# B&R Automation Studio project PLC code - cp
Automation Studio 4.1.4.357

## Configuration Dryer

CPU X20CP0483, AutomationRuntime G4.93, Build 4.1.2, Safety 0.0

### Task classes (Cpu.sw)
```
Cyclic#1 (cycle 8000 us, tolerance 8000 us):
  BasicDetec <- ExtPack._Media.BasicDetectMediaCtrl.BasicDetectMediaCtrl_v1.BasicDetectMediaCtrl.prg (BuildOptions=-D _IGNORE_CHECKLIB)
  ThickFast <- ExtPack._Media.ThicknessCtrl.ThicknessCtrl_v2.ThicknessCtrl_Fast.prg (BuildOptions=-D _IGNORE_CHECKLIB)
  VisuInks <- (binary) (BuildOptions=-D _IGNORE_CHECKLIB)
Cyclic#2 (cycle 12000 us, tolerance 24000 us):
  Initialize <- Dryer.Config.Initialize.prg (BuildOptions=-D _IGNORE_CHECKLIB)
  InitAxis <- ExtPack._Motion.AxisCtrl.AxisCtrl_v2.InitAxisControl.prg (BuildOptions=-D _IGNORE_CHECKLIB)
  Belt <- ExtPack._Motion.AxisCtrl.AxisCtrl_v2.AxisCtrl.prg (BuildOptions=-D _IGNORE_CHECKLIB)
  Elevation <- ExtPack._Motion.AxisCtrl.AxisCtrl_v2.AxisCtrl.prg (BuildOptions=-D _IGNORE_CHECKLIB)
  InitInvert <- ExtPack._Motion.InverterCtrl.InverterCtrl_v1.InitInverterCtrl.prg (BuildOptions=-D _IGNORE_CHECKLIB)
  Inverter1 <- ExtPack._Motion.InverterCtrl.InverterCtrl_v1.InverterCtrl.prg (BuildOptions=-D _IGNORE_CHECKLIB)
  Inverter2 <- ExtPack._Motion.InverterCtrl.InverterCtrl_v1.InverterCtrl.prg (BuildOptions=-D _IGNORE_CHECKLIB)
Cyclic#4 (cycle 32000 us, tolerance 96000 us):
  PhyInputs <- Dryer.PhysicalMapping.PhysicalMapInputs.prg (BuildOptions=-D _IGNORE_CHECKLIB)
  ThickCtrl <- ExtPack._Media.ThicknessCtrl.ThicknessCtrl_v2.ThicknessCtrl.prg (BuildOptions=-D _IGNORE_CHECKLIB)
  DryerFast <- Dryer.DryerCtrl.DryerCtrl_Fast.prg (BuildOptions=-D _IGNORE_CHECKLIB)
  BeltCtrl <- ExtPack._Transport.BeltCtrl.BeltCtrl_v1.BeltCtrl.prg (BuildOptions=-D _IGNORE_CHECKLIB)
  InitSimple <- ExtPack.SimpleBlockCtrl.SimpleBlockCtrl_v1.InitSimpleBlockCtrl.prg (BuildOptions=-D _IGNORE_CHECKLIB)
  SimpleBloc <- ExtPack.SimpleBlockCtrl.SimpleBlockCtrl_v1.SimpleBlockCtrl.prg (BuildOptions=-D _IGNORE_CHECKLIB)
  InitTransV <- ExtPack._Transport.TransVacuumCtrl.TransVacuumCtrl_v1.InitTransVacuumCtrl.prg (BuildOptions=-D _IGNORE_CHECKLIB)
  TransVacuu <- ExtPack._Transport.TransVacuumCtrl.TransVacuumCtrl_v1.TransVacuumCtrl.prg (BuildOptions=-D _IGNORE_CHECKLIB)
  InitJamDet <- ExtPack._Transport.JamDetectCtrl.JamDetect_v1.InitJamDetect.prg (BuildOptions=-D _IGNORE_CHECKLIB)
  JamDetect <- ExtPack._Transport.JamDetectCtrl.JamDetect_v1.JamDetect.prg (BuildOptions=-D _IGNORE_CHECKLIB)
  ArcLampGew <- ExtPack._Cure.ArcLampGEW.ArcLampGew_v1.ArcLampGewCtrl.prg (BuildOptions=-D _IGNORE_CHECKLIB)
  NIRAdphos <- ExtPack._Cure.NIRAdphos.NIRAdphos_v1.NIRAdphosCtrl.prg (BuildOptions=-D _IGNORE_CHECKLIB)
  HMI <- Dryer.HMI.HMI.prg (BuildOptions=-D _IGNORE_CHECKLIB)
  PhysOutput <- Dryer.PhysicalMapping.PhysicalMapOutputs.prg (BuildOptions=-D _IGNORE_CHECKLIB)
Cyclic#5 (cycle 80000 us, tolerance 160000 us):
  MachConfig <- Dryer.Config.MachineConfigurator.prg (BuildOptions=-D _IGNORE_CHECKLIB)
  DryerSlow <- Dryer.DryerCtrl.DryerCtrl_Slow.prg (BuildOptions=-D _IGNORE_CHECKLIB)
  ThickReadE <- ExtPack._Media.ThicknessCtrl.ThicknessCtrl_v2.ThickReadEnergy.prg (BuildOptions=-D _IGNORE_CHECKLIB)
  EventLogGe <- ExtPack._Tools.EventLog.EventLog_v1.EventLogGen.prg (BuildOptions=-D _IGNORE_CHECKLIB)
  SavePerman <- Dryer.Config.SavePermanent.prg (BuildOptions=-D _IGNORE_CHECKLIB)
NcDataObjects: AcpErrTxt <- AxisTables.AcpErrTxt.dob, acp10etxen <- AxisTables.acp10etxen.dob, BK1_S1400a <- AxisTables.BK1_S1400_a.dob, BK1_S1400i <- AxisTables.BK1_S1400_i.dob, BeltS1400a <- AxisTables.BeltS1400_a.dob, BeltS1400i <- AxisTables.BeltS1400_i.dob
Binaries: Acp10sys, udbdef, TCData, mvLoader, TCLang, arsvcreg, OpcUaSrv, acp10cfg, Acp10map, iomap, asfw, Role, ashwac, sysconf, ashwd, User, arconfig, EFIunits, EFIfunct, TC, gAlrHist, gAlrCore, OpcUaMap
Libraries: Acp10sdc, Acp10man, AsBrStr, Acp10par, NcGlobal, Acp10_MC, Acp10sim, sys_lib, brsystem, operator, runtime, astime, AsSafety, FileIO, standard, AsXml, asstring, AsFifo, MTTypes, MTFilter, MTBasics, AsTCP, AsIecCon, AsIOAcc, AsBrMath, AsEPL, ArEventLog, AsARCfg, ArProject, AsHttp, DataObj, FBs, Functions, ConvertFun, EvLogLib, BRSE_JSON, UtMgr, MpAlarmX, MpBase, MpCom, MpServer, AxisFunc, ThickLib, AsOpcUac, ErrACS380, arssl, aruser, powerlnk, assem, asopcuas, ascanopen
```

### Hardware
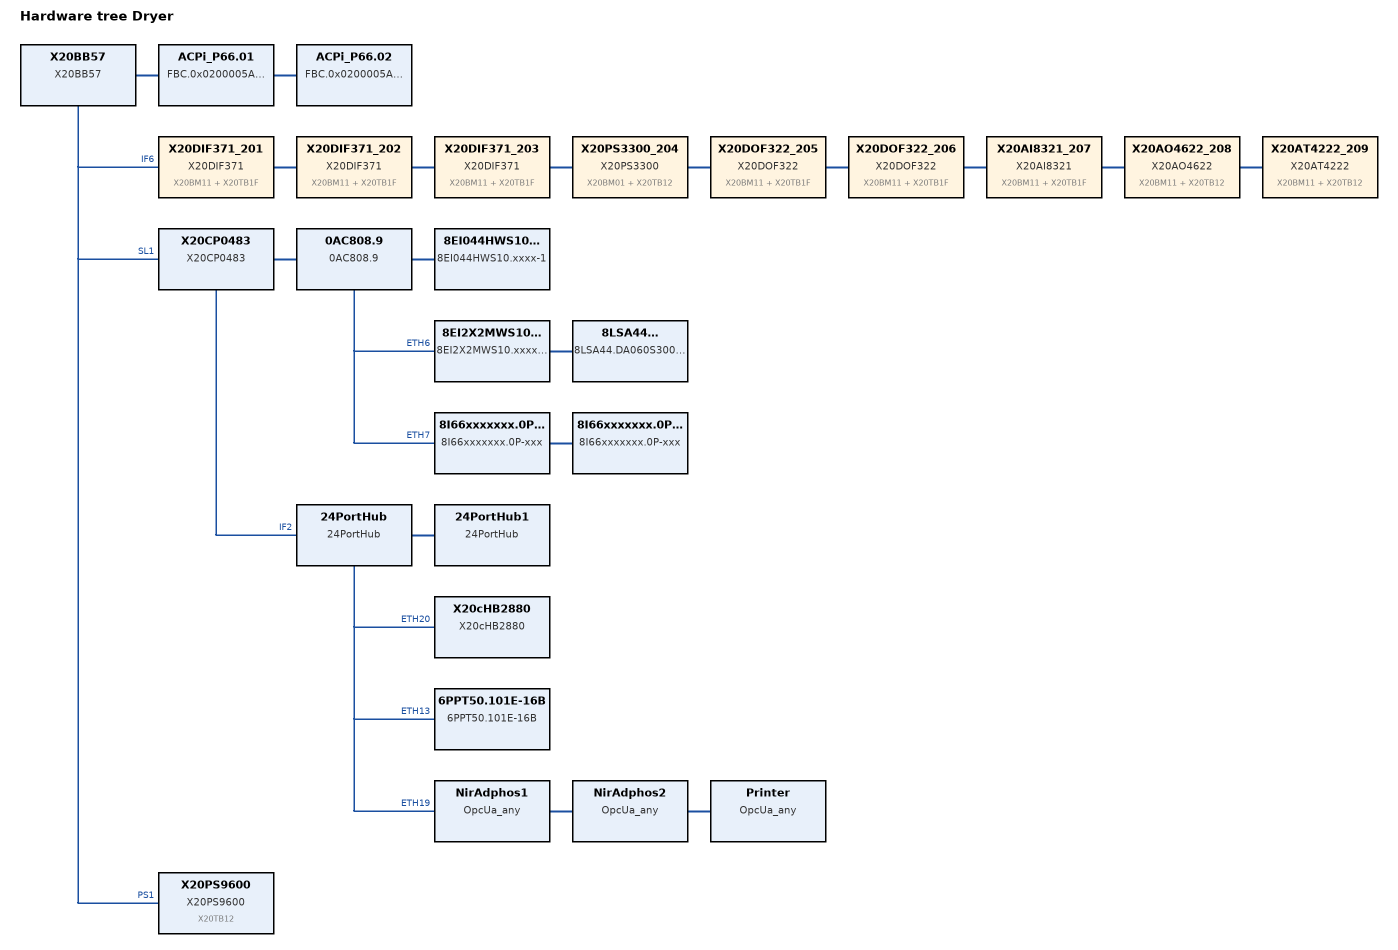
```
0AC808.9 : 0AC808.9 v1.0.0.0  [ETH1 -> X20CP0483.IF3 [Cable Type=PowerlinkCable, Length=10, Version=1.0.0.3]; ETH5 -> 8EI044HWS10.xxxx-1_BELT.PLK1 [Cable Type=PowerlinkCable, Length=10, Version=1.0.0.3]; ETH6 -> 8EI2X2MWS10.xxxx-1.PLK1 [Cable Type=PowerlinkCable, Length=10, Version=1.0.0.3]; ETH7 -> 8I66xxxxxxx.0P-81.PLK1 [Cable Type=PowerlinkCable, Length=10, Version=1.0.0.3]]
24PortHub : 24PortHub v1.0.0.1  [ETH7 -> X20CP0483.IF2 [Cable Type=PowerlinkCable, Length=10, Version=1.0.0.3]; ETH13 -> 6PPT50.101E-16B.ETH1 [Cable Type=PowerlinkCable, Length=10, Version=1.0.0.3]; ETH19 -> NirAdphos1.ETH1 [Cable Type=PowerlinkCable, Length=10, Version=1.0.0.3]; ETH20 -> X20cHB2880.ETH1 [Cable Type=PowerlinkCable, Length=10, Version=1.0.0.3]; ETH24 -> 24PortHub1.ETH3 [Cable Type=PowerlinkCable, Length=10, Version=1.0.0.3]]
24PortHub1 : 24PortHub v1.0.0.1  [ETH3 -> 24PortHub.ETH24 [Cable Type=PowerlinkCable, Length=10, Version=1.0.0.3]]
6PPT50.101E-16B : 6PPT50.101E-16B v1.3.8.0  [ETH1 -> 24PortHub.ETH13 [Cable Type=PowerlinkCable, Length=10, Version=1.0.0.3]]
  Terminal = true
  Startmode = 2
  ShowBootlogoWeb = 1
  Mode = Manual
  InternetAddress = 192.168.125.48
  Subnetmask = 255.255.255.0
  Hostname = efi_dryer_hmi
  Screensaver = 1
  Screensavertype = 0
  ActivateBuzzer = 1
  PasswordVNC = 
  SelectedFavoriteWeb = 192.168.125.47:81/index.html
  Favorites_Web1 = 
  BrowserVKeyboard = 0
  PasswordCIFS = 
  PasswordService = 
  ANSLAuthUserName = 
8EI044HWS10.xxxx-1_BELT : 8EI044HWS10.xxxx-1 v2.3.1.1  [PLK1 -> 0AC808.9.ETH5 [Cable Type=PowerlinkCable, Length=10, Version=1.0.0.3]]
  MotionTP = Acp10Arnc0
  Ax1Interface = Ax1EnDat
8EI2X2MWS10.xxxx-1 : 8EI2X2MWS10.xxxx-1 v2.3.1.1  [PLK1 -> 0AC808.9.ETH6 (NodeNumber=21) [Cable Type=PowerlinkCable, Length=10, Version=1.0.0.3]; EC1 -> 8LSA44.DA060S300-3.EC]
  MotionTP = Acp10Arnc0
  Ax1Interface = Ax1EnDat
8I66xxxxxxx.0P-81 : 8I66xxxxxxx.0P-xxx v2.5.1.0  [PLK1 -> 0AC808.9.ETH7 (NodeNumber=81) [Cable Type=PowerlinkCable, Length=10, Version=1.0.0.3]; PLK2 -> 8I66xxxxxxx.0P-82.PLK1 (NodeNumber=81) [Cable Type=PowerlinkCable, Length=10, Version=1.0.0.3]]
  FunctionModel = Standard
  Supervision = off
  UnitOfSetpoint = Rpm
  IOM_AIDP1 = LFT
  IOM_AIDP2 = LCR
  IOM_AIDP3 = OTRN
  IOM_AIDP4 = IL1R
  IOM_AIDP5 = AI1R
  IOM_AIDP6 = AI2R
  IOM_AIDP7 = AI3R
  IOM_AIDP8 = OL1I
  IOM_AIDP9 = AO1I
  IOM_R1ctrl = mapped
  IOM_R2ctrl = mapped
  IOM_LO1ctrl = mapped
  IOM_AO1ctrl = mapped
  Sel_AO1T = 0A
  Sel_NameplateMask = 8Ix6T401500_IEC
  Cfg_NSP = 2940
  Cfg_NCR = 277
  Cfg_COS = 82
  Sel_TUN = AUTO
8I66xxxxxxx.0P-82 : 8I66xxxxxxx.0P-xxx v2.5.1.0  [PLK1 -> 8I66xxxxxxx.0P-81.PLK2 [Cable Type=PowerlinkCable, Length=10, Version=1.0.0.3]]
  FunctionModel = Standard
  Supervision = off
  UnitOfSetpoint = Rpm
  IOM_AIDP1 = LFT
  IOM_AIDP2 = LCR
  IOM_AIDP3 = OTRN
  IOM_AIDP4 = IL1R
  IOM_AIDP5 = AI1R
  IOM_AIDP6 = AI2R
  IOM_AIDP7 = AI3R
  IOM_AIDP8 = OL1I
  IOM_AIDP9 = AO1I
  IOM_R1ctrl = mapped
  IOM_R2ctrl = mapped
  IOM_LO1ctrl = mapped
  IOM_AO1ctrl = mapped
  Sel_AO1T = 0A
  Sel_NameplateMask = 8Ix6T401500_IEC
  Cfg_NSP = 2940
  Cfg_NCR = 277
  Cfg_COS = 82
  Sel_TUN = AUTO
8LSA44.DA060S300-3 : 8LSA44.DA060S300-3 v1.0.10.37  [EC -> 8EI2X2MWS10.xxxx-1.EC1; MT -> 8EI2X2MWS10.xxxx-1.MT1]
ACPi_P66.01 : FBC.0x0200005A.320.ACPi_P66_P76 v1.3 (OrderNumber=ACPi_P66_P76)  [CAN1 -> X20BB57.IF7 (NodeNumber=81)]
  p2002sub5_connecttomaster = 2
  p2016sub3_connecttomaster = 1
  p2016subd_connecttomaster = 5
  p2016sub21_connecttomaster = 1
  p2016sub22_connecttomaster = 1
  p2016sub3e_connecttomaster = 5
  p2029sub16_connecttomaster = 2
  p2038sub2_connecttomaster = 4
  p2038sub3_connecttomaster = 4
  p2038sub4_connecttomaster = 2
  p2038sub5_connecttomaster = 2
  p203csub2_connecttomaster = 5
  p203csub3_connecttomaster = 5
  p6040_connecttomaster = 0
  p6041_connecttomaster = 0
  p6042_connecttomaster = 0
  p6044_connecttomaster = 0
  p6077_connecttomaster = 1
  p1800_transmissionselection = 2
  p1801_transmissionselection = 2
  p1802_transmissionselection = 2
ACPi_P66.02 : FBC.0x0200005A.320.ACPi_P66_P76 v1.3 (OrderNumber=ACPi_P66_P76)  [CAN1 -> ACPi_P66.01.CAN2]
  p2002sub5_connecttomaster = 2
  p2016sub3_connecttomaster = 1
  p2016subd_connecttomaster = 5
  p2016sub21_connecttomaster = 1
  p2016sub22_connecttomaster = 1
  p2016sub3e_connecttomaster = 5
  p2029sub16_connecttomaster = 2
  p2038sub2_connecttomaster = 4
  p2038sub3_connecttomaster = 4
  p2038sub4_connecttomaster = 2
  p2038sub5_connecttomaster = 2
  p203csub2_connecttomaster = 5
  p203csub3_connecttomaster = 5
  p6040_connecttomaster = 0
  p6041_connecttomaster = 0
  p6042_connecttomaster = 0
  p6044_connecttomaster = 0
  p6077_connecttomaster = 1
  p1800_transmissionselection = 2
  p1801_transmissionselection = 2
  p1802_transmissionselection = 2
NirAdphos1 : OpcUa_any v1.0.0.1  [ETH1 -> 24PortHub.ETH19 [Cable Type=PowerlinkCable, Length=10, Version=1.0.0.3]; ETH2 -> NirAdphos2.ETH1 [Cable Type=PowerlinkCable, Length=10, Version=1.0.0.3]]
  ServerDiagnostics = on
  ServerEndpointUrl = opc.tcp://192.168.125.91:4840
  PnPTimeout = 2500
  SecurityMsgMode = 0
  Channel1
  ChannelID1 = HMI
  ChannelBrowsePath1 = /0:Root/0:Objects/3:ServerInterfaces/4:SendData/4:DB11_HMI_out/4:HMI
  ChannelType1 = INT
  Channel2
  ChannelID2 = Hardware
  ChannelBrowsePath2 = /0:Root/0:Objects/3:ServerInterfaces/4:SendData/4:DB11_HMI_out/4:Hardware
  ChannelType2 = INT
  Channel3
  ChannelID3 = Software
  ChannelBrowsePath3 = /0:Root/0:Objects/3:ServerInterfaces/4:SendData/4:DB11_HMI_out/4:Software
  ChannelType3 = INT
  Channel4
  ChannelID4 = Interface
  ChannelBrowsePath4 = /0:Root/0:Objects/3:ServerInterfaces/4:SendData/4:DB11_HMI_out/4:interface
  ChannelType4 = INT
  Channel5
  ChannelID5 = NIRno
  ChannelBrowsePath5 = /0:Root/0:Objects/3:ServerInterfaces/4:SendData/4:DB11_HMI_out/4:general/4:NIRno
  ChannelType5 = INT
  Channel6
  ChannelID6 = NIRwidth
  ChannelBrowsePath6 = /0:Root/0:Objects/3:ServerInterfaces/4:SendData/4:DB11_HMI_out/4:general/4:NIRwidth
  ChannelType6 = INT
  Channel7
  ChannelID7 = calPower
  ChannelBrowsePath7 = /0:Root/0:Objects/3:ServerInterfaces/4:SendData/4:DB11_HMI_out/4:general/4:calPower
  ChannelType7 = INT
  Channel8
  ChannelID8 = speed
  ChannelBrowsePath8 = /0:Root/0:Objects/3:ServerInterfaces/4:SendData/4:DB11_HMI_out/4:general/4:speed
  ChannelType8 = REAL
  Channel9
  ChannelID9 = Watchdog1
  ChannelBrowsePath9 = /0:Root/0:Objects/3:ServerInterfaces/4:SendData/4:DB11_HMI_out/4:general/4:Watchdog
  Channel10
  ChannelID10 = EmFailNo_1
  ChannelBrowsePath10 = /0:Root/0:Objects/3:ServerInterfaces/4:SendData/4:DB11_HMI_out/4:module/4:[1]/4:EmFailNo
  ChannelType10 = USINT
  Channel11
  ChannelID11 = EmFailNo_2
  ChannelBrowsePath11 = /0:Root/0:Objects/3:ServerInterfaces/4:SendData/4:DB11_HMI_out/4:module/4:[2]/4:EmFailNo
  ChannelType11 = USINT
  Channel12
  ChannelID12 = ExhAirRunning_1
  ChannelBrowsePath12 = /0:Root/0:Objects/3:ServerInterfaces/4:SendData/4:DB11_HMI_out/4:module/4:[1]/4:ExhAirRunning
  Channel13
  ChannelID13 = ExhAirRunning_2
  ChannelBrowsePath13 = /0:Root/0:Objects/3:ServerInterfaces/4:SendData/4:DB11_HMI_out/4:module/4:[2]/4:ExhAirRunning
  Channel14
  ChannelID14 = NIRstatus_1
  ChannelBrowsePath14 = /0:Root/0:Objects/3:ServerInterfaces/4:SendData/4:DB11_HMI_out/4:module/4:[1]/4:NIRstatus
  ChannelType14 = INT
  Channel15
  ChannelID15 = NIRstatus_2
  ChannelBrowsePath15 = /0:Root/0:Objects/3:ServerInterfaces/4:SendData/4:DB11_HMI_out/4:module/4:[2]/4:NIRstatus
  ChannelType15 = INT
  Channel16
  ChannelID16 = airPressIn_1
  ChannelBrowsePath16 = /0:Root/0:Objects/3:ServerInterfaces/4:SendData/4:DB11_HMI_out/4:module/4:[1]/4:airPressIn
  ChannelType16 = REAL
  Channel17
  ChannelID17 = airPressIn_2
  ChannelBrowsePath17 = /0:Root/0:Objects/3:ServerInterfaces/4:SendData/4:DB11_HMI_out/4:module/4:[2]/4:airPressIn
  ChannelType17 = REAL
  Channel18
  ChannelID18 = airPressOut_1
  ChannelBrowsePath18 = /0:Root/0:Objects/3:ServerInterfaces/4:SendData/4:DB11_HMI_out/4:module/4:[1]/4:airPressOut
  ChannelType18 = REAL
  Channel19
  ChannelID19 = airPressOut_2
  ChannelBrowsePath19 = /0:Root/0:Objects/3:ServerInterfaces/4:SendData/4:DB11_HMI_out/4:module/4:[2]/4:airPressOut
  ChannelType19 = REAL
  Channel20
  ChannelID20 = airFilter_1
  ChannelBrowsePath20 = /0:Root/0:Objects/3:ServerInterfaces/4:SendData/4:DB11_HMI_out/4:module/4:[1]/4:airFilter
  ChannelType20 = INT
  Channel21
  ChannelID21 = airFilter_2
  ChannelBrowsePath21 = /0:Root/0:Objects/3:ServerInterfaces/4:SendData/4:DB11_HMI_out/4:module/4:[2]/4:airFilter
  ChannelType21 = INT
  Channel22
  ChannelID22 = actSpeedIn_1
  ChannelBrowsePath22 = /0:Root/0:Objects/3:ServerInterfaces/4:SendData/4:DB11_HMI_out/4:module/4:[1]/4:actSpeedIn
  ChannelType22 = INT
  Channel23
  ChannelID23 = actSpeedIn_2
  ChannelBrowsePath23 = /0:Root/0:Objects/3:ServerInterfaces/4:SendData/4:DB11_HMI_out/4:module/4:[2]/4:actSpeedIn
  ChannelType23 = INT
  Channel24
  ChannelID24 = actSpeedOut_1
  ChannelBrowsePath24 = /0:Root/0:Objects/3:ServerInterfaces/4:SendData/4:DB11_HMI_out/4:module/4:[1]/4:actSpeedOut
  ChannelType24 = INT
  Channel25
  ChannelID25 = actSpeedOut_2
  ChannelBrowsePath25 = /0:Root/0:Objects/3:ServerInterfaces/4:SendData/4:DB11_HMI_out/4:module/4:[2]/4:actSpeedOut
  ChannelType25 = INT
  Channel26
  ChannelID26 = actPower_1
  ChannelBrowsePath26 = /0:Root/0:Objects/3:ServerInterfaces/4:SendData/4:DB11_HMI_out/4:module/4:[1]/4:actPower
  ChannelType26 = INT
  Channel27
  ChannelID27 = actPower_2
  ChannelBrowsePath27 = /0:Root/0:Objects/3:ServerInterfaces/4:SendData/4:DB11_HMI_out/4:module/4:[2]/4:actPower
  ChannelType27 = INT
  Channel28
  ChannelID28 = Watchdog2
  ChannelBrowsePath28 = /0:Root/0:Objects/3:ServerInterfaces/4:SendData/4:DB11_HMI_out/4:general/4:Watchdog
  Channel29
  ChannelID29 = Reset
  ChannelBrowsePath29 = /0:Root/0:Objects/3:ServerInterfaces/5:RecData/5:DB10_HMI_in/5:reset
  ChannelDirection29 = OUT
  Channel30
  ChannelID30 = Pend
  ChannelBrowsePath30 = /0:Root/0:Objects/3:ServerInterfaces/5:RecData/5:DB10_HMI_in/5:product/5:Pend
  ChannelDirection30 = OUT
  ChannelType30 = REAL
  Channel31
  ChannelID31 = Pstart
  ChannelBrowsePath31 = /0:Root/0:Objects/3:ServerInterfaces/5:RecData/5:DB10_HMI_in/5:product/5:Pstart
  ChannelDirection31 = OUT
  ChannelType31 = REAL
  Channel32
  ChannelID32 = Vend
  ChannelBrowsePath32 = /0:Root/0:Objects/3:ServerInterfaces/5:RecData/5:DB10_HMI_in/5:product/5:Vend
  ChannelDirection32 = OUT
  ChannelType32 = REAL
  Channel33
  ChannelID33 = Vstart
  ChannelBrowsePath33 = /0:Root/0:Objects/3:ServerInterfaces/5:RecData/5:DB10_HMI_in/5:product/5:Vstart
  ChannelDirection33 = OUT
  ChannelType33 = REAL
  Channel34
  ChannelID34 = AdjPos
  ChannelBrowsePath34 = /0:Root/0:Objects/3:ServerInterfaces/5:RecData/5:DB10_HMI_in/5:product/5:adjPos
  ChannelDirection34 = OUT
  ChannelType34 = INT
  Channel35
  ChannelID35 = WebWidth
  ChannelBrowsePath35 = /0:Root/0:Objects/3:ServerInterfaces/5:RecData/5:DB10_HMI_in/5:product/5:webWidth
  ChannelDirection35 = OUT
  ChannelType35 = INT
  Channel36
  ChannelID36 = Adjust_1
  ChannelBrowsePath36 = /0:Root/0:Objects/3:ServerInterfaces/5:RecData/5:DB10_HMI_in/5:module/5:[1]/5:adjust
  ChannelDirection36 = OUT
  ChannelType36 = INT
  Channel37
  ChannelID37 = Adjust_2
  ChannelBrowsePath37 = /0:Root/0:Objects/3:ServerInterfaces/5:RecData/5:DB10_HMI_in/5:module/5:[2]/5:adjust
  ChannelDirection37 = OUT
  ChannelType37 = INT
  Channel38
  ChannelID38 = EnableMod_1
  ChannelBrowsePath38 = /0:Root/0:Objects/3:ServerInterfaces/5:RecData/5:DB10_HMI_in/5:module/5:[1]/5:enableMod
  ChannelDirection38 = OUT
  Channel39
  ChannelID39 = EnableMod_2
  ChannelBrowsePath39 = /0:Root/0:Objects/3:ServerInterfaces/5:RecData/5:DB10_HMI_in/5:module/5:[2]/5:enableMod
  ChannelDirection39 = OUT
  Channel40
  ChannelID40 = WatchdogOut
  ChannelBrowsePath40 = /0:Root/0:Objects/3:ServerInterfaces/5:RecData/5:DB10_HMI_in/5:Watchdog
  ChannelDirection40 = OUT
  Channel41
  ChannelID41 = Enable_DDC
  ChannelBrowsePath41 = /0:Root/0:Objects/3:ServerInterfaces/5:RecData/5:DB10_HMI_in/5:DDCon
  ChannelDirection41 = OUT
  Channel42
  ChannelID42 = NIR1_Int1
  ChannelBrowsePath42 = /0:Root/0:Objects/3:ServerInterfaces/5:RecData/5:DB10_HMI_in/5:intensity/5:intensity/5:[1]
  ChannelDirection42 = OUT
  ChannelType42 = INT
  Channel43
  ChannelID43 = NIR1_Int2
  ChannelBrowsePath43 = /0:Root/0:Objects/3:ServerInterfaces/5:RecData/5:DB10_HMI_in/5:intensity/5:intensity/5:[2]
  ChannelDirection43 = OUT
  ChannelType43 = INT
  Channel44
  ChannelID44 = NIR1_Int3
  ChannelBrowsePath44 = /0:Root/0:Objects/3:ServerInterfaces/5:RecData/5:DB10_HMI_in/5:intensity/5:intensity/5:[3]
  ChannelDirection44 = OUT
  ChannelType44 = INT
  Channel45
  ChannelID45 = NIR1_Int4
  ChannelBrowsePath45 = /0:Root/0:Objects/3:ServerInterfaces/5:RecData/5:DB10_HMI_in/5:intensity/5:intensity/5:[4]
  ChannelDirection45 = OUT
  ChannelType45 = INT
  Channel46
  ChannelID46 = NIR1_Int5
  ChannelBrowsePath46 = /0:Root/0:Objects/3:ServerInterfaces/5:RecData/5:DB10_HMI_in/5:intensity/5:intensity/5:[5]
  ChannelDirection46 = OUT
  ChannelType46 = INT
  Channel47
  ChannelID47 = NIR1_Int6
  ChannelBrowsePath47 = /0:Root/0:Objects/3:ServerInterfaces/5:RecData/5:DB10_HMI_in/5:intensity/5:intensity/5:[6]
  ChannelDirection47 = OUT
  ChannelType47 = INT
  Channel48
  ChannelID48 = NIR1_Int7
  ChannelBrowsePath48 = /0:Root/0:Objects/3:ServerInterfaces/5:RecData/5:DB10_HMI_in/5:intensity/5:intensity/5:[7]
  ChannelDirection48 = OUT
  ChannelType48 = INT
  Channel49
  ChannelID49 = NIR1_Int8
  ChannelBrowsePath49 = /0:Root/0:Objects/3:ServerInterfaces/5:RecData/5:DB10_HMI_in/5:intensity/5:intensity/5:[8]
  ChannelDirection49 = OUT
  ChannelType49 = INT
  Channel50
  ChannelID50 = NIR1_Int9
  ChannelBrowsePath50 = /0:Root/0:Objects/3:ServerInterfaces/5:RecData/5:DB10_HMI_in/5:intensity/5:intensity/5:[9]
  ChannelDirection50 = OUT
  ChannelType50 = INT
  Channel51
  ChannelID51 = NIR1_Int10
  ChannelBrowsePath51 = /0:Root/0:Objects/3:ServerInterfaces/5:RecData/5:DB10_HMI_in/5:intensity/5:intensity/5:[10]
  ChannelDirection51 = OUT
  ChannelType51 = INT
  Channel52
  ChannelID52 = NIR1_Int11
  ChannelBrowsePath52 = /0:Root/0:Objects/3:ServerInterfaces/5:RecData/5:DB10_HMI_in/5:intensity/5:intensity/5:[11]
  ChannelDirection52 = OUT
  ChannelType52 = INT
  Channel53
  ChannelID53 = NIR1_Int12
  ChannelBrowsePath53 = /0:Root/0:Objects/3:ServerInterfaces/5:RecData/5:DB10_HMI_in/5:intensity/5:intensity/5:[12]
  ChannelDirection53 = OUT
  ChannelType53 = INT
  Channel54
  ChannelID54 = NIR1_Int13
  ChannelBrowsePath54 = /0:Root/0:Objects/3:ServerInterfaces/5:RecData/5:DB10_HMI_in/5:intensity/5:intensity/5:[13]
  ChannelDirection54 = OUT
  ChannelType54 = INT
  Channel55
  ChannelID55 = NIR1_Int14
  ChannelBrowsePath55 = /0:Root/0:Objects/3:ServerInterfaces/5:RecData/5:DB10_HMI_in/5:intensity/5:intensity/5:[14]
  ChannelDirection55 = OUT
  ChannelType55 = INT
  Channel56
  ChannelID56 = NIR1_Int15
  ChannelBrowsePath56 = /0:Root/0:Objects/3:ServerInterfaces/5:RecData/5:DB10_HMI_in/5:intensity/5:intensity/5:[15]
  ChannelDirection56 = OUT
  ChannelType56 = INT
  Channel57
  ChannelID57 = NIR1_Int16
  ChannelBrowsePath57 = /0:Root/0:Objects/3:ServerInterfaces/5:RecData/5:DB10_HMI_in/5:intensity/5:intensity/5:[16]
  ChannelDirection57 = OUT
  ChannelType57 = INT
  Channel58
  ChannelID58 = NIR1_Int17
  ChannelBrowsePath58 = /0:Root/0:Objects/3:ServerInterfaces/5:RecData/5:DB10_HMI_in/5:intensity/5:intensity/5:[17]
  ChannelDirection58 = OUT
  ChannelType58 = INT
  Channel59
  ChannelID59 = NIR1_Int18
  ChannelBrowsePath59 = /0:Root/0:Objects/3:ServerInterfaces/5:RecData/5:DB10_HMI_in/5:intensity/5:intensity/5:[18]
  ChannelDirection59 = OUT
  ChannelType59 = INT
  Channel60
  ChannelID60 = NIR1_Int19
  ChannelBrowsePath60 = /0:Root/0:Objects/3:ServerInterfaces/5:RecData/5:DB10_HMI_in/5:intensity/5:intensity/5:[19]
  ChannelDirection60 = OUT
  ChannelType60 = INT
  Channel61
  ChannelID61 = NIR1_Int20
  ChannelBrowsePath61 = /0:Root/0:Objects/3:ServerInterfaces/5:RecData/5:DB10_HMI_in/5:intensity/5:intensity/5:[20]
  ChannelDirection61 = OUT
  ChannelType61 = INT
  Channel62
  ChannelID62 = NIR1_Int21
  ChannelBrowsePath62 = /0:Root/0:Objects/3:ServerInterfaces/5:RecData/5:DB10_HMI_in/5:intensity/5:intensity/5:[21]
  ChannelDirection62 = OUT
  ChannelType62 = INT
  Channel63
  ChannelID63 = NIR1_Int22
  ChannelBrowsePath63 = /0:Root/0:Objects/3:ServerInterfaces/5:RecData/5:DB10_HMI_in/5:intensity/5:intensity/5:[22]
  ChannelDirection63 = OUT
  ChannelType63 = INT
  Channel64
  ChannelID64 = NIR1_Int23
  ChannelBrowsePath64 = /0:Root/0:Objects/3:ServerInterfaces/5:RecData/5:DB10_HMI_in/5:intensity/5:intensity/5:[23]
  ChannelDirection64 = OUT
  ChannelType64 = INT
  Channel65
  ChannelID65 = NIR1_Int24
  ChannelBrowsePath65 = /0:Root/0:Objects/3:ServerInterfaces/5:RecData/5:DB10_HMI_in/5:intensity/5:intensity/5:[24]
  ChannelDirection65 = OUT
  ChannelType65 = INT
  Channel66
  ChannelID66 = NIR1_Int25
  ChannelBrowsePath66 = /0:Root/0:Objects/3:ServerInterfaces/5:RecData/5:DB10_HMI_in/5:intensity/5:intensity/5:[25]
  ChannelDirection66 = OUT
  ChannelType66 = INT
  Channel67
  ChannelID67 = NIR1_Int26
  ChannelBrowsePath67 = /0:Root/0:Objects/3:ServerInterfaces/5:RecData/5:DB10_HMI_in/5:intensity/5:intensity/5:[26]
  ChannelDirection67 = OUT
  ChannelType67 = INT
  Channel68
  ChannelID68 = NIR1_Int27
  ChannelBrowsePath68 = /0:Root/0:Objects/3:ServerInterfaces/5:RecData/5:DB10_HMI_in/5:intensity/5:intensity/5:[27]
  ChannelDirection68 = OUT
  ChannelType68 = INT
  Channel69
  ChannelID69 = NIR1_Int28
  ChannelBrowsePath69 = /0:Root/0:Objects/3:ServerInterfaces/5:RecData/5:DB10_HMI_in/5:intensity/5:intensity/5:[28]
  ChannelDirection69 = OUT
  ChannelType69 = INT
  Channel70
  ChannelID70 = NIR1_Int29
  ChannelBrowsePath70 = /0:Root/0:Objects/3:ServerInterfaces/5:RecData/5:DB10_HMI_in/5:intensity/5:intensity/5:[29]
  ChannelDirection70 = OUT
  ChannelType70 = INT
  Channel71
  ChannelID71 = NIR1_Int30
  ChannelBrowsePath71 = /0:Root/0:Objects/3:ServerInterfaces/5:RecData/5:DB10_HMI_in/5:intensity/5:intensity/5:[30]
  ChannelDirection71 = OUT
  ChannelType71 = INT
  Channel72
  ChannelID72 = NIR1_Int31
  ChannelBrowsePath72 = /0:Root/0:Objects/3:ServerInterfaces/5:RecData/5:DB10_HMI_in/5:intensity/5:intensity/5:[31]
  ChannelDirection72 = OUT
  ChannelType72 = INT
  Channel73
  ChannelID73 = NIR1_Int32
  ChannelBrowsePath73 = /0:Root/0:Objects/3:ServerInterfaces/5:RecData/5:DB10_HMI_in/5:intensity/5:intensity/5:[32]
  ChannelDirection73 = OUT
  ChannelType73 = INT
  Channel74
  ChannelID74 = NIR1_Int33
  ChannelBrowsePath74 = /0:Root/0:Objects/3:ServerInterfaces/5:RecData/5:DB10_HMI_in/5:intensity/5:intensity/5:[33]
  ChannelDirection74 = OUT
  ChannelType74 = INT
  Channel75
  ChannelID75 = NIR1_Int34
  ChannelBrowsePath75 = /0:Root/0:Objects/3:ServerInterfaces/5:RecData/5:DB10_HMI_in/5:intensity/5:intensity/5:[34]
  ChannelDirection75 = OUT
  ChannelType75 = INT
  Channel76
  ChannelID76 = NIR1_Int35
  ChannelBrowsePath76 = /0:Root/0:Objects/3:ServerInterfaces/5:RecData/5:DB10_HMI_in/5:intensity/5:intensity/5:[35]
  ChannelDirection76 = OUT
  ChannelType76 = INT
  Channel77
  ChannelID77 = NIR1_Int36
  ChannelBrowsePath77 = /0:Root/0:Objects/3:ServerInterfaces/5:RecData/5:DB10_HMI_in/5:intensity/5:intensity/5:[36]
  ChannelDirection77 = OUT
  ChannelType77 = INT
  Channel78
  ChannelID78 = NIR1_Int37
  ChannelBrowsePath78 = /0:Root/0:Objects/3:ServerInterfaces/5:RecData/5:DB10_HMI_in/5:intensity/5:intensity/5:[37]
  ChannelDirection78 = OUT
  ChannelType78 = INT
  Channel79
  ChannelID79 = NIR1_Int38
  ChannelBrowsePath79 = /0:Root/0:Objects/3:ServerInterfaces/5:RecData/5:DB10_HMI_in/5:intensity/5:intensity/5:[38]
  ChannelDirection79 = OUT
  ChannelType79 = INT
  Channel80
  ChannelID80 = NIR1_Int39
  ChannelBrowsePath80 = /0:Root/0:Objects/3:ServerInterfaces/5:RecData/5:DB10_HMI_in/5:intensity/5:intensity/5:[39]
  ChannelDirection80 = OUT
  ChannelType80 = INT
  Channel81
  ChannelID81 = NIR1_Int40
  ChannelBrowsePath81 = /0:Root/0:Objects/3:ServerInterfaces/5:RecData/5:DB10_HMI_in/5:intensity/5:intensity/5:[40]
  ChannelDirection81 = OUT
  ChannelType81 = INT
  Channel82
  ChannelID82 = NIR1_Int41
  ChannelBrowsePath82 = /0:Root/0:Objects/3:ServerInterfaces/5:RecData/5:DB10_HMI_in/5:intensity/5:intensity/5:[41]
  ChannelDirection82 = OUT
  ChannelType82 = INT
  Channel83
  ChannelID83 = NIR1_Int42
  ChannelBrowsePath83 = /0:Root/0:Objects/3:ServerInterfaces/5:RecData/5:DB10_HMI_in/5:intensity/5:intensity/5:[42]
  ChannelDirection83 = OUT
  ChannelType83 = INT
  Channel84
  ChannelID84 = NIR1_Int43
  ChannelBrowsePath84 = /0:Root/0:Objects/3:ServerInterfaces/5:RecData/5:DB10_HMI_in/5:intensity/5:intensity/5:[43]
  ChannelDirection84 = OUT
  ChannelType84 = INT
  Channel85
  ChannelID85 = NIR1_Int44
  ChannelBrowsePath85 = /0:Root/0:Objects/3:ServerInterfaces/5:RecData/5:DB10_HMI_in/5:intensity/5:intensity/5:[44]
  ChannelDirection85 = OUT
  ChannelType85 = INT
  Channel86
  ChannelID86 = NIR1_Int45
  ChannelBrowsePath86 = /0:Root/0:Objects/3:ServerInterfaces/5:RecData/5:DB10_HMI_in/5:intensity/5:intensity/5:[45]
  ChannelDirection86 = OUT
  ChannelType86 = INT
  Channel87
  ChannelID87 = NIR1_Int46
  ChannelBrowsePath87 = /0:Root/0:Objects/3:ServerInterfaces/5:RecData/5:DB10_HMI_in/5:intensity/5:intensity/5:[46]
  ChannelDirection87 = OUT
  ChannelType87 = INT
  Channel88
  ChannelID88 = NIR1_Int47
  ChannelBrowsePath88 = /0:Root/0:Objects/3:ServerInterfaces/5:RecData/5:DB10_HMI_in/5:intensity/5:intensity/5:[47]
  ChannelDirection88 = OUT
  ChannelType88 = INT
  Channel89
  ChannelID89 = NIR1_Int48
  ChannelBrowsePath89 = /0:Root/0:Objects/3:ServerInterfaces/5:RecData/5:DB10_HMI_in/5:intensity/5:intensity/5:[48]
  ChannelDirection89 = OUT
  ChannelType89 = INT
NirAdphos2 : OpcUa_any v1.0.0.1  [ETH1 -> NirAdphos1.ETH2 [Cable Type=PowerlinkCable, Length=10, Version=1.0.0.3]; ETH2 -> Printer.ETH1 [Cable Type=PowerlinkCable, Length=10, Version=1.0.0.3]]
  ServerDiagnostics = on
  ServerEndpointUrl = opc.tcp://192.168.125.92:4840
  PnPTimeout = 2500
  SecurityMsgMode = 0
  Channel1
  ChannelID1 = NIR2_Int1
  ChannelBrowsePath1 = /0:Root/0:Objects/3:ServerInterfaces/0:RecData/4:DB10_HMI_in/4:intensity/4:[1]
  ChannelDirection1 = OUT
  ChannelType1 = INT
  Channel2
  ChannelID2 = NIR2_Int2
  ChannelBrowsePath2 = /0:Root/0:Objects/3:ServerInterfaces/0:RecData/4:DB10_HMI_in/4:intensity/4:[2]
  ChannelDirection2 = OUT
  ChannelType2 = INT
  Channel3
  ChannelID3 = NIR2_Int3
  ChannelBrowsePath3 = /0:Root/0:Objects/3:ServerInterfaces/0:RecData/4:DB10_HMI_in/4:intensity/4:[3]
  ChannelDirection3 = OUT
  ChannelType3 = INT
  Channel4
  ChannelID4 = NIR2_Int4
  ChannelBrowsePath4 = /0:Root/0:Objects/3:ServerInterfaces/0:RecData/4:DB10_HMI_in/4:intensity/4:[4]
  ChannelDirection4 = OUT
  ChannelType4 = INT
  Channel5
  ChannelID5 = NIR2_Int5
  ChannelBrowsePath5 = /0:Root/0:Objects/3:ServerInterfaces/0:RecData/4:DB10_HMI_in/4:intensity/4:[5]
  ChannelDirection5 = OUT
  ChannelType5 = INT
  Channel6
  ChannelID6 = NIR2_Int6
  ChannelBrowsePath6 = /0:Root/0:Objects/3:ServerInterfaces/0:RecData/4:DB10_HMI_in/4:intensity/4:[6]
  ChannelDirection6 = OUT
  ChannelType6 = INT
  Channel7
  ChannelID7 = NIR2_Int7
  ChannelBrowsePath7 = /0:Root/0:Objects/3:ServerInterfaces/0:RecData/4:DB10_HMI_in/4:intensity/4:[7]
  ChannelDirection7 = OUT
  ChannelType7 = INT
  Channel8
  ChannelID8 = NIR2_Int8
  ChannelBrowsePath8 = /0:Root/0:Objects/3:ServerInterfaces/0:RecData/4:DB10_HMI_in/4:intensity/4:[8]
  ChannelDirection8 = OUT
  ChannelType8 = INT
  Channel9
  ChannelID9 = NIR2_Int9
  ChannelBrowsePath9 = /0:Root/0:Objects/3:ServerInterfaces/0:RecData/4:DB10_HMI_in/4:intensity/4:[9]
  ChannelDirection9 = OUT
  ChannelType9 = INT
  Channel10
  ChannelID10 = NIR2_Int10
  ChannelBrowsePath10 = /0:Root/0:Objects/3:ServerInterfaces/0:RecData/4:DB10_HMI_in/4:intensity/4:[10]
  ChannelDirection10 = OUT
  ChannelType10 = INT
  Channel11
  ChannelID11 = NIR2_Int11
  ChannelBrowsePath11 = /0:Root/0:Objects/3:ServerInterfaces/0:RecData/4:DB10_HMI_in/4:intensity/4:[11]
  ChannelDirection11 = OUT
  ChannelType11 = INT
  Channel12
  ChannelID12 = NIR2_Int12
  ChannelBrowsePath12 = /0:Root/0:Objects/3:ServerInterfaces/0:RecData/4:DB10_HMI_in/4:intensity/4:[12]
  ChannelDirection12 = OUT
  ChannelType12 = INT
  Channel13
  ChannelID13 = NIR2_Int13
  ChannelBrowsePath13 = /0:Root/0:Objects/3:ServerInterfaces/0:RecData/4:DB10_HMI_in/4:intensity/4:[13]
  ChannelDirection13 = OUT
  ChannelType13 = INT
  Channel14
  ChannelID14 = NIR2_Int14
  ChannelBrowsePath14 = /0:Root/0:Objects/3:ServerInterfaces/0:RecData/4:DB10_HMI_in/4:intensity/4:[14]
  ChannelDirection14 = OUT
  ChannelType14 = INT
  Channel15
  ChannelID15 = NIR2_Int15
  ChannelBrowsePath15 = /0:Root/0:Objects/3:ServerInterfaces/0:RecData/4:DB10_HMI_in/4:intensity/4:[15]
  ChannelDirection15 = OUT
  ChannelType15 = INT
  Channel16
  ChannelID16 = NIR2_Int16
  ChannelBrowsePath16 = /0:Root/0:Objects/3:ServerInterfaces/0:RecData/4:DB10_HMI_in/4:intensity/4:[16]
  ChannelDirection16 = OUT
  ChannelType16 = INT
  Channel17
  ChannelID17 = NIR2_Int17
  ChannelBrowsePath17 = /0:Root/0:Objects/3:ServerInterfaces/0:RecData/4:DB10_HMI_in/4:intensity/4:[17]
  ChannelDirection17 = OUT
  ChannelType17 = INT
  Channel18
  ChannelID18 = NIR2_Int18
  ChannelBrowsePath18 = /0:Root/0:Objects/3:ServerInterfaces/0:RecData/4:DB10_HMI_in/4:intensity/4:[18]
  ChannelDirection18 = OUT
  ChannelType18 = INT
  Channel19
  ChannelID19 = NIR2_Int19
  ChannelBrowsePath19 = /0:Root/0:Objects/3:ServerInterfaces/0:RecData/4:DB10_HMI_in/4:intensity/4:[19]
  ChannelDirection19 = OUT
  ChannelType19 = INT
  Channel20
  ChannelID20 = NIR2_Int20
  ChannelBrowsePath20 = /0:Root/0:Objects/3:ServerInterfaces/0:RecData/4:DB10_HMI_in/4:intensity/4:[20]
  ChannelDirection20 = OUT
  ChannelType20 = INT
  Channel21
  ChannelID21 = NIR2_Int21
  ChannelBrowsePath21 = /0:Root/0:Objects/3:ServerInterfaces/0:RecData/4:DB10_HMI_in/4:intensity/4:[21]
  ChannelDirection21 = OUT
  ChannelType21 = INT
  Channel22
  ChannelID22 = NIR2_Int22
  ChannelBrowsePath22 = /0:Root/0:Objects/3:ServerInterfaces/0:RecData/4:DB10_HMI_in/4:intensity/4:[22]
  ChannelDirection22 = OUT
  ChannelType22 = INT
  Channel23
  ChannelID23 = NIR2_Int23
  ChannelBrowsePath23 = /0:Root/0:Objects/3:ServerInterfaces/0:RecData/4:DB10_HMI_in/4:intensity/4:[23]
  ChannelDirection23 = OUT
  ChannelType23 = INT
  Channel24
  ChannelID24 = NIR2_Int24
  ChannelBrowsePath24 = /0:Root/0:Objects/3:ServerInterfaces/0:RecData/4:DB10_HMI_in/4:intensity/4:[24]
  ChannelDirection24 = OUT
  ChannelType24 = INT
  Channel25
  ChannelID25 = NIR2_Int25
  ChannelBrowsePath25 = /0:Root/0:Objects/3:ServerInterfaces/0:RecData/4:DB10_HMI_in/4:intensity/4:[25]
  ChannelDirection25 = OUT
  ChannelType25 = INT
  Channel26
  ChannelID26 = NIR2_Int26
  ChannelBrowsePath26 = /0:Root/0:Objects/3:ServerInterfaces/0:RecData/4:DB10_HMI_in/4:intensity/4:[26]
  ChannelDirection26 = OUT
  ChannelType26 = INT
  Channel27
  ChannelID27 = NIR2_Int27
  ChannelBrowsePath27 = /0:Root/0:Objects/3:ServerInterfaces/0:RecData/4:DB10_HMI_in/4:intensity/4:[27]
  ChannelDirection27 = OUT
  ChannelType27 = INT
  Channel28
  ChannelID28 = NIR2_Int28
  ChannelBrowsePath28 = /0:Root/0:Objects/3:ServerInterfaces/0:RecData/4:DB10_HMI_in/4:intensity/4:[28]
  ChannelDirection28 = OUT
  ChannelType28 = INT
  Channel29
  ChannelID29 = NIR2_Int29
  ChannelBrowsePath29 = /0:Root/0:Objects/3:ServerInterfaces/0:RecData/4:DB10_HMI_in/4:intensity/4:[29]
  ChannelDirection29 = OUT
  ChannelType29 = INT
  Channel30
  ChannelID30 = NIR2_Int30
  ChannelBrowsePath30 = /0:Root/0:Objects/3:ServerInterfaces/0:RecData/4:DB10_HMI_in/4:intensity/4:[30]
  ChannelDirection30 = OUT
  ChannelType30 = INT
  Channel31
  ChannelID31 = NIR2_Int31
  ChannelBrowsePath31 = /0:Root/0:Objects/3:ServerInterfaces/0:RecData/4:DB10_HMI_in/4:intensity/4:[31]
  ChannelDirection31 = OUT
  ChannelType31 = INT
  Channel32
  ChannelID32 = NIR2_Int32
  ChannelBrowsePath32 = /0:Root/0:Objects/3:ServerInterfaces/0:RecData/4:DB10_HMI_in/4:intensity/4:[32]
  ChannelDirection32 = OUT
  ChannelType32 = INT
  Channel33
  ChannelID33 = NIR2_Int33
  ChannelBrowsePath33 = /0:Root/0:Objects/3:ServerInterfaces/0:RecData/4:DB10_HMI_in/4:intensity/4:[33]
  ChannelDirection33 = OUT
  ChannelType33 = INT
  Channel34
  ChannelID34 = NIR2_Int34
  ChannelBrowsePath34 = /0:Root/0:Objects/3:ServerInterfaces/0:RecData/4:DB10_HMI_in/4:intensity/4:[34]
  ChannelDirection34 = OUT
  ChannelType34 = INT
  Channel35
  ChannelID35 = NIR2_Int35
  ChannelBrowsePath35 = /0:Root/0:Objects/3:ServerInterfaces/0:RecData/4:DB10_HMI_in/4:intensity/4:[35]
  ChannelDirection35 = OUT
  ChannelType35 = INT
  Channel36
  ChannelID36 = NIR2_Int36
  ChannelBrowsePath36 = /0:Root/0:Objects/3:ServerInterfaces/0:RecData/4:DB10_HMI_in/4:intensity/4:[36]
  ChannelDirection36 = OUT
  ChannelType36 = INT
  Channel37
  ChannelID37 = NIR2_Int37
  ChannelBrowsePath37 = /0:Root/0:Objects/3:ServerInterfaces/0:RecData/4:DB10_HMI_in/4:intensity/4:[37]
  ChannelDirection37 = OUT
  ChannelType37 = INT
  Channel38
  ChannelID38 = NIR2_Int38
  ChannelBrowsePath38 = /0:Root/0:Objects/3:ServerInterfaces/0:RecData/4:DB10_HMI_in/4:intensity/4:[38]
  ChannelDirection38 = OUT
  ChannelType38 = INT
  Channel39
  ChannelID39 = NIR2_Int39
  ChannelBrowsePath39 = /0:Root/0:Objects/3:ServerInterfaces/0:RecData/4:DB10_HMI_in/4:intensity/4:[39]
  ChannelDirection39 = OUT
  ChannelType39 = INT
  Channel40
  ChannelID40 = NIR2_Int40
  ChannelBrowsePath40 = /0:Root/0:Objects/3:ServerInterfaces/0:RecData/4:DB10_HMI_in/4:intensity/4:[40]
  ChannelDirection40 = OUT
  ChannelType40 = INT
  Channel41
  ChannelID41 = NIR2_Int41
  ChannelBrowsePath41 = /0:Root/0:Objects/3:ServerInterfaces/0:RecData/4:DB10_HMI_in/4:intensity/4:[41]
  ChannelDirection41 = OUT
  ChannelType41 = INT
  Channel42
  ChannelID42 = NIR2_Int42
  ChannelBrowsePath42 = /0:Root/0:Objects/3:ServerInterfaces/0:RecData/4:DB10_HMI_in/4:intensity/4:[42]
  ChannelDirection42 = OUT
  ChannelType42 = INT
  Channel43
  ChannelID43 = NIR2_Int43
  ChannelBrowsePath43 = /0:Root/0:Objects/3:ServerInterfaces/0:RecData/4:DB10_HMI_in/4:intensity/4:[43]
  ChannelDirection43 = OUT
  ChannelType43 = INT
  Channel44
  ChannelID44 = NIR2_Int44
  ChannelBrowsePath44 = /0:Root/0:Objects/3:ServerInterfaces/0:RecData/4:DB10_HMI_in/4:intensity/4:[44]
  ChannelDirection44 = OUT
  ChannelType44 = INT
  Channel45
  ChannelID45 = NIR2_Int45
  ChannelBrowsePath45 = /0:Root/0:Objects/3:ServerInterfaces/0:RecData/4:DB10_HMI_in/4:intensity/4:[45]
  ChannelDirection45 = OUT
  ChannelType45 = INT
  Channel46
  ChannelID46 = NIR2_Int46
  ChannelBrowsePath46 = /0:Root/0:Objects/3:ServerInterfaces/0:RecData/4:DB10_HMI_in/4:intensity/4:[46]
  ChannelDirection46 = OUT
  ChannelType46 = INT
  Channel47
  ChannelID47 = NIR2_Int47
  ChannelBrowsePath47 = /0:Root/0:Objects/3:ServerInterfaces/0:RecData/4:DB10_HMI_in/4:intensity/4:[47]
  ChannelDirection47 = OUT
  ChannelType47 = INT
  Channel48
  ChannelID48 = NIR2_Int48
  ChannelBrowsePath48 = /0:Root/0:Objects/3:ServerInterfaces/0:RecData/4:DB10_HMI_in/4:intensity/4:[48]
  ChannelDirection48 = OUT
  ChannelType48 = INT
Printer : OpcUa_any v1.0.0.1  [ETH1 -> NirAdphos2.ETH2 [Cable Type=PowerlinkCable, Length=10, Version=1.0.0.3]]
  ServerDiagnostics = on
  ServerEndpointUrl = opc.tcp://192.168.125.10:4840
  UserIdentifyToken = 1
  Username = PressCore
  Password = h98o76
  Channel1
  ChannelID1 = xRunTransport
  ChannelBrowsePath1 = /0:Root/0:Objects/4:PLC/4:Modules/6:&:&:/6:Global PV/6:gDryerRemoteData/6:Commands/6:xRunTransport
  Channel2
  ChannelID2 = xPrepareToDry
  ChannelBrowsePath2 = /0:Root/0:Objects/4:PLC/4:Modules/6:&:&:/6:Global PV/6:gDryerRemoteData/6:Commands/6:xPrepareToDry
  ChannelSamplingInterval2 = 200
  ChannelPublishingInterval2 = 400
  Channel3
  ChannelID3 = xStartDrying
  ChannelBrowsePath3 = /0:Root/0:Objects/4:PLC/4:Modules/6:&:&:/6:Global PV/6:gDryerRemoteData/6:Commands/6:xStartDrying
  ChannelSamplingInterval3 = 200
  ChannelPublishingInterval3 = 400
  Channel4
  ChannelID4 = xEnableNir
  ChannelBrowsePath4 = /0:Root/0:Objects/4:PLC/4:Modules/6:&:&:/6:Global PV/6:gDryerRemoteData/6:Parameters/6:xEnableNir
  ChannelSamplingInterval4 = 200
  ChannelPublishingInterval4 = 400
  Channel5
  ChannelID5 = xEnableArcLampDrying
  ChannelBrowsePath5 = /0:Root/0:Objects/4:PLC/4:Modules/6:&:&:/6:Global PV/6:gDryerRemoteData/6:Parameters/6:xEnableArcLamp
  ChannelSamplingInterval5 = 200
  ChannelPublishingInterval5 = 400
  Channel6
  ChannelID6 = rBeltSpeedSetPoint
  ChannelBrowsePath6 = /0:Root/0:Objects/4:PLC/4:Modules/6:&:&:/6:Global PV/6:gDryerRemoteData/6:Parameters/6:rBeltSpeedSetPoint
  ChannelType6 = REAL
  Channel7
  ChannelID7 = rBoardLength
  ChannelBrowsePath7 = /0:Root/0:Objects/4:PLC/4:Modules/6:&:&:/6:Global PV/6:gDryerRemoteData/6:Parameters/6:Media/6:rLength
  ChannelSamplingInterval7 = 200
  ChannelPublishingInterval7 = 400
  ChannelType7 = REAL
  Channel8
  ChannelID8 = rBoardWidth
  ChannelBrowsePath8 = /0:Root/0:Objects/4:PLC/4:Modules/6:&:&:/6:Global PV/6:gDryerRemoteData/6:Parameters/6:Media/6:rWidth
  ChannelSamplingInterval8 = 200
  ChannelPublishingInterval8 = 400
  ChannelType8 = REAL
  Channel9
  ChannelID9 = rBoardThickness
  ChannelBrowsePath9 = /0:Root/0:Objects/4:PLC/4:Modules/6:&:&:/6:Global PV/6:gDryerRemoteData/6:Parameters/6:Media/6:rThickness
  ChannelSamplingInterval9 = 200
  ChannelPublishingInterval9 = 400
  ChannelType9 = REAL
  Channel10
  ChannelID10 = rBoardGap
  ChannelBrowsePath10 = /0:Root/0:Objects/4:PLC/4:Modules/6:&:&:/6:Global PV/6:gDryerRemoteData/6:Parameters/6:Media/6:rGap
  ChannelSamplingInterval10 = 200
  ChannelPublishingInterval10 = 400
  ChannelType10 = REAL
  Channel11
  ChannelID11 = Signals_xMediaPresent
  ChannelBrowsePath11 = /0:Root/0:Objects/4:PLC/4:Modules/6:&:&:/6:Global PV/6:gDryerRemoteData/6:Signals/6:xMediaPresent
  ChannelSamplingInterval11 = 200
  ChannelPublishingInterval11 = 400
  Channel12
  ChannelID12 = Signals_xBreakerOKBlowerInput
  ChannelBrowsePath12 = /0:Root/0:Objects/4:PLC/4:Modules/6:&:&:/6:Global PV/6:gDryerRemoteData/6:Signals/6:xBreakerOKBlowerInput
  ChannelSamplingInterval12 = 200
  ChannelPublishingInterval12 = 400
  Channel13
  ChannelID13 = Signals_xBreakerOKBlowerOutput
  ChannelBrowsePath13 = /0:Root/0:Objects/4:PLC/4:Modules/6:&:&:/6:Global PV/6:gDryerRemoteData/6:Signals/6:xBreakerOKBlowerOutput
  ChannelSamplingInterval13 = 200
  ChannelPublishingInterval13 = 400
  Channel14
  ChannelID14 = Signals_Safety_xMovementsEnabled
  ChannelBrowsePath14 = /0:Root/0:Objects/4:PLC/4:Modules/6:&:&:/6:Global PV/6:gDryerRemoteData/6:Signals/6:Safety/6:xMovementsEnabled
  ChannelSamplingInterval14 = 200
  ChannelPublishingInterval14 = 400
  Channel15
  ChannelID15 = Signals_Safety_xRemoteEStopOK
  ChannelBrowsePath15 = /0:Root/0:Objects/4:PLC/4:Modules/6:&:&:/6:Global PV/6:gDryerRemoteData/6:Signals/6:Safety/6:xRemoteEStopOK
  ChannelSamplingInterval15 = 200
  ChannelPublishingInterval15 = 400
  Channel16
  ChannelID16 = Signals_Safety_xEStopFrontOK
  ChannelBrowsePath16 = /0:Root/0:Objects/4:PLC/4:Modules/6:&:&:/6:Global PV/6:gDryerRemoteData/6:Signals/6:Safety/6:xEStopFrontOK
  ChannelSamplingInterval16 = 200
  ChannelPublishingInterval16 = 400
  Channel17
  ChannelID17 = Signals_Safety_xEStopRearOK
  ChannelBrowsePath17 = /0:Root/0:Objects/4:PLC/4:Modules/6:&:&:/6:Global PV/6:gDryerRemoteData/6:Signals/6:Safety/6:xEStopRearOK
  ChannelSamplingInterval17 = 200
  ChannelPublishingInterval17 = 400
  Channel18
  ChannelID18 = Signals_Safety_xClosedFrontIn
  ChannelBrowsePath18 = /0:Root/0:Objects/4:PLC/4:Modules/6:&:&:/6:Global PV/6:gDryerRemoteData/6:Signals/6:Safety/6:xClosedFrontInput
  ChannelSamplingInterval18 = 200
  ChannelPublishingInterval18 = 400
  Channel19
  ChannelID19 = Signals_Safety_xClosedFrontOut
  ChannelBrowsePath19 = /0:Root/0:Objects/4:PLC/4:Modules/6:&:&:/6:Global PV/6:gDryerRemoteData/6:Signals/6:Safety/6:xClosedFrontOutput
  ChannelSamplingInterval19 = 200
  ChannelPublishingInterval19 = 400
  Channel20
  ChannelID20 = Signals_Safety_xClosedRearIn
  ChannelBrowsePath20 = /0:Root/0:Objects/4:PLC/4:Modules/6:&:&:/6:Global PV/6:gDryerRemoteData/6:Signals/6:Safety/6:xClosedRearInput
  ChannelSamplingInterval20 = 200
  ChannelPublishingInterval20 = 400
  Channel21
  ChannelID21 = Signals_Safety_xClosedRearOut
  ChannelBrowsePath21 = /0:Root/0:Objects/4:PLC/4:Modules/6:&:&:/6:Global PV/6:gDryerRemoteData/6:Signals/6:Safety/6:xClosedRearOutput
  ChannelSamplingInterval21 = 200
  ChannelPublishingInterval21 = 400
  Channel22
  ChannelID22 = rDocumentWidth
  ChannelBrowsePath22 = /0:Root/0:Objects/4:PLC/4:Modules/6:&:&:/6:Global PV/6:gDryerRemoteData/6:Parameters/6:Media/6:rDocWidth
  ChannelSamplingInterval22 = 200
  ChannelPublishingInterval22 = 400
  ChannelType22 = REAL
  Channel23
  ChannelID23 = rDocumentLength
  ChannelBrowsePath23 = /0:Root/0:Objects/4:PLC/4:Modules/6:&:&:/6:Global PV/6:gDryerRemoteData/6:Parameters/6:Media/6:rDocLength
  ChannelSamplingInterval23 = 200
  ChannelPublishingInterval23 = 400
  ChannelType23 = REAL
  Channel24
  ChannelID24 = xLineEmptyingBelt
  ChannelBrowsePath24 = /0:Root/0:Objects/4:PLC/4:Modules/6:&:&:/6:Global PV/6:gDryerRemoteData/6:Parameters/6:xLineEmptyingBelt
  ChannelSamplingInterval24 = 200
  ChannelPublishingInterval24 = 400
  Channel25
  ChannelID25 = xPrepareToEmptyBelt
  ChannelBrowsePath25 = /0:Root/0:Objects/4:PLC/4:Modules/6:&:&:/6:Global PV/6:gDryerRemoteData/6:Commands/6:xPrepareToEmptyBelt
  ChannelSamplingInterval25 = 200
  ChannelPublishingInterval25 = 400
  Channel26
  ChannelID26 = rDocumentOffset
  ChannelBrowsePath26 = /0:Root/0:Objects/4:PLC/4:Modules/6:&:&:/6:Global PV/6:gDryerRemoteData/6:Parameters/6:Media/6:rDocCrossOffset
  ChannelSamplingInterval26 = 200
  ChannelPublishingInterval26 = 400
  ChannelType26 = REAL
  Channel27
  ChannelID27 = rCrossOffset
  ChannelBrowsePath27 = /0:Root/0:Objects/4:PLC/4:Modules/6:&:&:/6:Global PV/6:gDryerRemoteData/6:Parameters/6:Media/6:rCrossOffset
  ChannelSamplingInterval27 = 200
  ChannelPublishingInterval27 = 400
  ChannelType27 = REAL
  Channel28
  ChannelID28 = rSubstratePowerReduction
  ChannelBrowsePath28 = /0:Root/0:Objects/4:PLC/4:Modules/6:&:&:/6:Global PV/6:gDryerRemoteData/6:Parameters/6:rSubstratePowerReduction
  ChannelSamplingInterval28 = 200
  ChannelPublishingInterval28 = 400
  ChannelType28 = REAL
  Channel29
  ChannelID29 = xEnableDDC
  ChannelBrowsePath29 = /0:Root/0:Objects/4:PLC/4:Modules/6:&:&:/6:Global PV/6:gDryerRemoteData/6:Parameters/6:xEnableDDC
  ChannelSamplingInterval29 = 200
  ChannelPublishingInterval29 = 400
  Channel30
  ChannelID30 = xPrinterBeltRuning
  ChannelBrowsePath30 = /0:Root/0:Objects/4:PLC/4:Modules/6:&:&:/6:Global PV/6:gDryerRemoteData/6:Parameters/6:xPrinterBeltRuning
  ChannelSamplingInterval30 = 200
  ChannelPublishingInterval30 = 400
X20AI8321_207 : X20AI8321 v1.5.0.0  [SS1 -> X20TB1F5.SS; SL -> X20BM11e.SL1]
  Supervision = off
  LowerLimit = -8192
  ChannelType01 = 4 to 20mA
  ChannelType02 = 4 to 20mA
  ChannelType03 = 4 to 20mA
  ChannelType04 = 4 to 20mA
  ChannelType05 = 4 to 20mA
  ChannelType06 = 4 to 20mA
  ChannelType07 = 4 to 20mA
  ChannelType08 = 4 to 20mA
X20AO4622_208 : X20AO4622 v1.3.0.0  [SS1 -> X20TB12b.SS; SL -> X20BM11f.SL1]
  Supervision = off
X20AT4222_209 : X20AT4222 v1.4.0.0  [SS1 -> X20TB12c.SS; SL -> X20BM11g.SL1]
  FunctionModel = FunctionModel001
  Supervision = off
  SensorType03 = off
  SensorType04 = off
X20BB57 : X20BB57 v1.2.0.0
  Connector IF7:
    Baudrate = 250000
    ActivateCanOpen = 1
    p100c_parametervalue = 1000
    p100d_parametervalue = 3
X20BM01 : X20BM01 v2.2.0.0  [X2X1 -> X20BM11b.X2X2]
X20BM11 : X20BM11 v1.1.0.0  [X2X1 -> X20BB57.IF6]
X20BM11a : X20BM11 v1.1.0.0  [X2X1 -> X20BM11.X2X2]
X20BM11b : X20BM11 v1.1.0.0  [X2X1 -> X20BM11a.X2X2]
X20BM11c : X20BM11 v1.1.0.0  [X2X1 -> X20BM01.X2X2]
X20BM11d : X20BM11 v1.1.0.0  [X2X1 -> X20BM11c.X2X2]
X20BM11e : X20BM11 v1.1.0.0  [X2X1 -> X20BM11d.X2X2]
X20BM11f : X20BM11 v1.1.0.0  [X2X1 -> X20BM11e.X2X2]
X20BM11g : X20BM11 v1.1.0.0  [X2X1 -> X20BM11f.X2X2]
X20CP0483 : X20CP0483 v1.6.0.0  [SL -> X20BB57.SL1]
  Connector IF2:
    ActivateDevice = 1
    HostName = efi_dryer
    Mode = Manual
    InternetAddress = 192.168.125.47
    SubnetMask = 255.255.255.0
    InaNodeNumber = 0
    ActivateSnmp = 2
  Connector IF3:
    DNAConfiguration = manual
    EplNatSubnet = 192.168.102.0
  ConfigurationID = Dryer
  UserPartitionSize = 0
  SimulationIPAddress = 192.168.0.138
  SimulationModeOpcUa = off
  PermanentPvSize = 5000
  RemanentGlobalPvSize = 10000
  VolatileGlobalPvSize = 1500000
  UserLoggerSize = 4096000
  EnableUsbRemoteInstall = 1
  EnableCfRemoteInstall = 1
  RebootReset = 1
  TimerDeviceType = EPLX2X
  TimerDevice = X20CP0483.IF3
  TaskClassIdleTime = 4000
  CyclicTaskClassCount = 6
  Cyclic1Duration = 8000
  Cyclic1Tolerance = 8000
  Cyclic1Stack = 16384
  Cyclic1Output = 1
  Cyclic2Duration = 12000
  Cyclic2Tolerance = 24000
  Cyclic2Stack = 16384
  Cyclic3Duration = 16000
  Cyclic3Tolerance = 48000
  Cyclic3Stack = 16384
  Cyclic4Duration = 32000
  Cyclic4Tolerance = 96000
  Cyclic4Stack = 16384
  Cyclic5Duration = 80000
  Cyclic5Tolerance = 160000
  Cyclic5Stack = 16384
  Cyclic6Duration = 88000
  Cyclic6Tolerance = 528000
  Cyclic7Duration = 1000000
  Cyclic7Tolerance = 1000000
  Cyclic8Duration = 800000
  Cyclic8Tolerance = 30400000
  FileDevice1
  FileDeviceName1 = USER
  FileDevicePath1 = USER_PATH
  FtpUser1
  FtpUsername1 = EFI  // EFI
  FtpUserPassword1 = 7G5n+wCoc8AAtJwOeMqQrBZ1Z+2KeIxeQkt+7Ofj72s=  // Castellon
  FtpUserSalt1 = xa1UK9Qk
  FTPAccessRight1 = 0
  FTPdevice1 = ALL
  ActivateOpcUa = 1
  OpcUaInformationModels_PV_Version = 2
  OpcUaInformationModel_Facet = 0
  OpcUaInformationModel_TypeInformation = 0
  OpcUaInformationModel_BaseObjectTypeForStructures = 0
X20DIF371_201 : X20DIF371 v1.3.0.0  [SS1 -> X20TB1F.SS; SL -> X20BM11.SL1]
  Supervision = off
X20DIF371_202 : X20DIF371 v1.3.0.0  [SS1 -> X20TB1F1.SS; SL -> X20BM11a.SL1]
  Supervision = off
X20DIF371_203 : X20DIF371 v1.3.0.0  [SS1 -> X20TB1F2.SS; SL -> X20BM11b.SL1]
  Supervision = off
X20DOF322_205 : X20DOF322 v1.5.0.0  [SS1 -> X20TB1F3.SS; SL -> X20BM11c.SL1]
  Supervision = off
X20DOF322_206 : X20DOF322 v1.5.0.0  [SS1 -> X20TB1F4.SS; SL -> X20BM11d.SL1]
  Supervision = off
X20PS3300_204 : X20PS3300 v1.4.0.0  [SS1 -> X20TB12a.SS; SL -> X20BM01.SL1]
  Supervision = off
X20PS9600 : X20PS9600 v1.6.0.0  [PS -> X20BB57.PS1; SS1 -> X20TB12.SS]
  Supervision = off
X20TB12 : X20TB12 v1.0.0.0
X20TB12a : X20TB12 v1.0.0.0
X20TB12b : X20TB12 v1.0.0.0
X20TB12c : X20TB12 v1.0.0.0
X20TB1F : X20TB1F v1.0.0.0
X20TB1F1 : X20TB1F v1.0.0.0
X20TB1F2 : X20TB1F v1.0.0.0
X20TB1F3 : X20TB1F v1.0.0.0
X20TB1F4 : X20TB1F v1.0.0.0
X20TB1F5 : X20TB1F v1.0.0.0
X20cHB2880 : X20cHB2880 v1.2.0.0  [ETH1 -> 24PortHub.ETH20 [Cable Type=PowerlinkCable, Length=10, Version=1.0.0.3]]
```

### IoMap.iom - X20CP0483/IoMap.iom
```iecst
VAR_CONFIG
	::gInverterSignalsPowerLink[1].In.ModuleOk AT %IX."8I66xxxxxxx.0P-81".ModuleOk;
	::gInverterSignalsPowerLink[1].In.StatusWord AT %IW."8I66xxxxxxx.0P-81".ETAD_Input;
	::gInverterSignalsPowerLink[1].Out.ControlWord AT %QW."8I66xxxxxxx.0P-81".CMDD_Output;
	::gInverterSignalsPowerLink[1].Out.SetSpeed AT %QW."8I66xxxxxxx.0P-81".LFRD_Output;
	::gInverterSignalsPowerLink[2].In.ModuleOk AT %IX."8I66xxxxxxx.0P-82".ModuleOk;
	::gInverterSignalsPowerLink[2].In.StatusWord AT %IW."8I66xxxxxxx.0P-82".ETAD_Input;
	::gInverterSignalsPowerLink[2].Out.ControlWord AT %QW."8I66xxxxxxx.0P-82".CMDD_Output;
	::gInverterSignalsPowerLink[2].Out.SetSpeed AT %QW."8I66xxxxxxx.0P-82".LFRD_Output;
	::X20DIF371_201.ModuleOk AT %IX."X20DIF371_201".ModuleOk;
	::X20DIF371_201.DInput[1] AT %IX."X20DIF371_201".DigitalInput01;
	::X20DIF371_201.DInput[2] AT %IX."X20DIF371_201".DigitalInput02;
	::X20DIF371_201.DInput[3] AT %IX."X20DIF371_201".DigitalInput03;
	::X20DIF371_201.DInput[4] AT %IX."X20DIF371_201".DigitalInput04;
	::X20DIF371_201.DInput[5] AT %IX."X20DIF371_201".DigitalInput05;
	::X20DIF371_201.DInput[6] AT %IX."X20DIF371_201".DigitalInput06;
	::X20DIF371_201.DInput[7] AT %IX."X20DIF371_201".DigitalInput07;
	::X20DIF371_201.DInput[8] AT %IX."X20DIF371_201".DigitalInput08;
	::X20DIF371_201.DInput[9] AT %IX."X20DIF371_201".DigitalInput09;
	::X20DIF371_201.DInput[10] AT %IX."X20DIF371_201".DigitalInput10;
	::X20DIF371_201.DInput[11] AT %IX."X20DIF371_201".DigitalInput11;
	::X20DIF371_201.DInput[12] AT %IX."X20DIF371_201".DigitalInput12;
	::X20DIF371_201.DInput[13] AT %IX."X20DIF371_201".DigitalInput13;
	::X20DIF371_201.DInput[14] AT %IX."X20DIF371_201".DigitalInput14;
	::X20DIF371_201.DInput[15] AT %IX."X20DIF371_201".DigitalInput15;
	::X20DIF371_201.DInput[16] AT %IX."X20DIF371_201".DigitalInput16;
	::X20DIF371_202.ModuleOk AT %IX."X20DIF371_202".ModuleOk;
	::X20DIF371_202.DInput[1] AT %IX."X20DIF371_202".DigitalInput01;
	::X20DIF371_202.DInput[2] AT %IX."X20DIF371_202".DigitalInput02;
	::X20DIF371_202.DInput[3] AT %IX."X20DIF371_202".DigitalInput03;
	::X20DIF371_202.DInput[4] AT %IX."X20DIF371_202".DigitalInput04;
	::X20DIF371_202.DInput[5] AT %IX."X20DIF371_202".DigitalInput05;
	::X20DIF371_202.DInput[6] AT %IX."X20DIF371_202".DigitalInput06;
	::X20DIF371_202.DInput[7] AT %IX."X20DIF371_202".DigitalInput07;
	::X20DIF371_202.DInput[8] AT %IX."X20DIF371_202".DigitalInput08;
	::X20DIF371_202.DInput[9] AT %IX."X20DIF371_202".DigitalInput09;
	::X20DIF371_202.DInput[10] AT %IX."X20DIF371_202".DigitalInput10;
	::X20DIF371_202.DInput[11] AT %IX."X20DIF371_202".DigitalInput11;
	::X20DIF371_202.DInput[12] AT %IX."X20DIF371_202".DigitalInput12;
	::X20DIF371_202.DInput[13] AT %IX."X20DIF371_202".DigitalInput13;
	::X20DIF371_202.DInput[14] AT %IX."X20DIF371_202".DigitalInput14;
	::X20DIF371_202.DInput[15] AT %IX."X20DIF371_202".DigitalInput15;
	::X20DIF371_202.DInput[16] AT %IX."X20DIF371_202".DigitalInput16;
	::X20DIF371_203.ModuleOk AT %IX."X20DIF371_203".ModuleOk;
	::X20DIF371_203.DInput[1] AT %IX."X20DIF371_203".DigitalInput01;
	::X20DIF371_203.DInput[2] AT %IX."X20DIF371_203".DigitalInput02;
	::X20DIF371_203.DInput[3] AT %IX."X20DIF371_203".DigitalInput03;
	::X20DIF371_203.DInput[4] AT %IX."X20DIF371_203".DigitalInput04;
	::X20DIF371_203.DInput[5] AT %IX."X20DIF371_203".DigitalInput05;
	::X20DIF371_203.DInput[6] AT %IX."X20DIF371_203".DigitalInput06;
	::X20DIF371_203.DInput[7] AT %IX."X20DIF371_203".DigitalInput07;
	::X20DIF371_203.DInput[8] AT %IX."X20DIF371_203".DigitalInput08;
	::X20DIF371_203.DInput[9] AT %IX."X20DIF371_203".DigitalInput09;
	::X20DIF371_203.DInput[10] AT %IX."X20DIF371_203".DigitalInput10;
	::X20DIF371_203.DInput[11] AT %IX."X20DIF371_203".DigitalInput11;
	::X20DIF371_203.DInput[12] AT %IX."X20DIF371_203".DigitalInput12;
	::X20DIF371_203.DInput[13] AT %IX."X20DIF371_203".DigitalInput13;
	::X20DIF371_203.DInput[14] AT %IX."X20DIF371_203".DigitalInput14;
	::X20DIF371_203.DInput[15] AT %IX."X20DIF371_203".DigitalInput15;
	::X20DIF371_203.DInput[16] AT %IX."X20DIF371_203".DigitalInput16;
	::X20DOF322_205.ModuleOk AT %IX."X20DOF322_205".ModuleOk;
	::X20DOF322_205.DOutput[1] AT %QX."X20DOF322_205".DigitalOutput01;
	::X20DOF322_205.DOutput[2] AT %QX."X20DOF322_205".DigitalOutput02;
	::X20DOF322_205.DOutput[3] AT %QX."X20DOF322_205".DigitalOutput03;
	::X20DOF322_205.DOutput[4] AT %QX."X20DOF322_205".DigitalOutput04;
	::X20DOF322_205.DOutput[5] AT %QX."X20DOF322_205".DigitalOutput05;
	::X20DOF322_205.DOutput[6] AT %QX."X20DOF322_205".DigitalOutput06;
	::X20DOF322_205.DOutput[7] AT %QX."X20DOF322_205".DigitalOutput07;
	::X20DOF322_205.DOutput[8] AT %QX."X20DOF322_205".DigitalOutput08;
	::X20DOF322_205.DOutput[9] AT %QX."X20DOF322_205".DigitalOutput09;
	::X20DOF322_205.DOutput[10] AT %QX."X20DOF322_205".DigitalOutput10;
	::X20DOF322_205.DOutput[11] AT %QX."X20DOF322_205".DigitalOutput11;
	::X20DOF322_205.DOutput[12] AT %QX."X20DOF322_205".DigitalOutput12;
	::X20DOF322_205.DOutput[13] AT %QX."X20DOF322_205".DigitalOutput13;
	::X20DOF322_205.DOutput[14] AT %QX."X20DOF322_205".DigitalOutput14;
	::X20DOF322_205.DOutput[15] AT %QX."X20DOF322_205".DigitalOutput15;
	::X20DOF322_205.DOutput[16] AT %QX."X20DOF322_205".DigitalOutput16;
	::X20DOF322_206.ModuleOk AT %IX."X20DOF322_206".ModuleOk;
	::X20DOF322_206.DOutput[1] AT %QX."X20DOF322_206".DigitalOutput01;
	::X20DOF322_206.DOutput[2] AT %QX."X20DOF322_206".DigitalOutput02;
	::X20DOF322_206.DOutput[3] AT %QX."X20DOF322_206".DigitalOutput03;
	::X20DOF322_206.DOutput[4] AT %QX."X20DOF322_206".DigitalOutput04;
	::X20DOF322_206.DOutput[5] AT %QX."X20DOF322_206".DigitalOutput05;
	::X20DOF322_206.DOutput[6] AT %QX."X20DOF322_206".DigitalOutput06;
	::X20DOF322_206.DOutput[7] AT %QX."X20DOF322_206".DigitalOutput07;
	::X20DOF322_206.DOutput[8] AT %QX."X20DOF322_206".DigitalOutput08;
	::X20DOF322_206.DOutput[9] AT %QX."X20DOF322_206".DigitalOutput09;
	::X20DOF322_206.DOutput[10] AT %QX."X20DOF322_206".DigitalOutput10;
	::X20DOF322_206.DOutput[11] AT %QX."X20DOF322_206".DigitalOutput11;
	::X20DOF322_206.DOutput[12] AT %QX."X20DOF322_206".DigitalOutput12;
	::X20DOF322_206.DOutput[13] AT %QX."X20DOF322_206".DigitalOutput13;
	::X20DOF322_206.DOutput[14] AT %QX."X20DOF322_206".DigitalOutput14;
	::X20DOF322_206.DOutput[15] AT %QX."X20DOF322_206".DigitalOutput15;
	::X20DOF322_206.DOutput[16] AT %QX."X20DOF322_206".DigitalOutput16;
	::X20AI8321_207.ModuleOk AT %IX."X20AI8321_207".ModuleOk;
	::X20AI8321_207.AInput[1] AT %IW."X20AI8321_207".AnalogInput01;
	::X20AI8321_207.AInput[2] AT %IW."X20AI8321_207".AnalogInput02;
	::X20AI8321_207.AInput[3] AT %IW."X20AI8321_207".AnalogInput03;
	::X20AI8321_207.AInput[4] AT %IW."X20AI8321_207".AnalogInput04;
	::X20AI8321_207.AInput[5] AT %IW."X20AI8321_207".AnalogInput05;
	::X20AI8321_207.AInput[6] AT %IW."X20AI8321_207".AnalogInput06;
	::X20AI8321_207.AInput[7] AT %IW."X20AI8321_207".AnalogInput07;
	::X20AI8321_207.AInput[8] AT %IW."X20AI8321_207".AnalogInput08;
	::X20AO4622_208.ModuleOk AT %IX."X20AO4622_208".ModuleOk;
	::X20AO4622_208.AOutput[1] AT %QW."X20AO4622_208".AnalogOutput01;
	::X20AO4622_208.AOutput[2] AT %QW."X20AO4622_208".AnalogOutput02;
	::X20AO4622_208.AOutput[3] AT %QW."X20AO4622_208".AnalogOutput03;
	::X20AO4622_208.AOutput[4] AT %QW."X20AO4622_208".AnalogOutput04;
	::X20AT4222_209.ModuleOk AT %IX."X20AT4222_209".ModuleOk;
	::X20AT4222_209.TempInput[1] AT %IW."X20AT4222_209".Temperature01;
	::X20AT4222_209.TempInput[2] AT %IW."X20AT4222_209".Temperature02;
	::X20AT4222_209.TempInput[3] AT %IW."X20AT4222_209".Temperature03;
	::X20AT4222_209.TempInput[4] AT %IW."X20AT4222_209".Temperature04;
	::gNirAdphos.Parameters.Comms.Pend AT %QD."NirAdphos1".Pend;
	::gNirAdphos.Parameters.Comms.Pstart AT %QD."NirAdphos1".Pstart;
	::gNirAdphos.Parameters.Comms.Vend AT %QD."NirAdphos1".Vend;
	::gNirAdphos.Parameters.Comms.Vstart AT %QD."NirAdphos1".Vstart;
	::gNirAdphos.Parameters.Comms.AdjPos AT %QW."NirAdphos1".AdjPos;
	::gNirAdphos.Parameters.Comms.WebWidth AT %QW."NirAdphos1".WebWidth;
	::gNirAdphos.Parameters.Comms.Modules[1].Adjust AT %QW."NirAdphos1".Adjust_1;
	::gNirAdphos.Parameters.Comms.Modules[2].Adjust AT %QW."NirAdphos1".Adjust_2;
	::gNirAdphos.Parameters.Comms.Modules[1].EnableMod AT %QX."NirAdphos1".EnableMod_1;
	::gNirAdphos.Parameters.Comms.Modules[2].EnableMod AT %QX."NirAdphos1".EnableMod_2;
	::gNirAdphos.Commands.xReset AT %QX."NirAdphos1".Reset;
	::gNirAdphos.Status.Comms.Version.HMI AT %IW."NirAdphos1".HMI;
	::gNirAdphos.Status.Comms.Version.Hardware AT %IW."NirAdphos1".Hardware;
	::gNirAdphos.Status.Comms.Version.Software AT %IW."NirAdphos1".Software;
	::gNirAdphos.Status.Comms.Version.Interface AT %IW."NirAdphos1".Interface;
	::gNirAdphos.Status.Comms.NirTotalActive AT %IW."NirAdphos1".NIRno;
	::gNirAdphos.Status.Comms.NirTotalActive AT %IX."NirAdphos1".NIRwidth;
	::gNirAdphos.Status.Comms.NirTotalActive AT %IX."NirAdphos1".calPower;
	::gNirAdphos.Status.Comms.NirWidth AT %IW."NirAdphos1".NIRwidth;
	::gNirAdphos.Status.Comms.CalPower AT %IW."NirAdphos1".calPower;
	::gNirAdphos.Status.Comms.Speed AT %ID."NirAdphos1".speed;
	::gNirAdphos.Status.Comms.Modules[1].ExtAirRunning AT %IX."NirAdphos1".ExhAirRunning_1;
	::gNirAdphos.Status.Comms.Modules[2].ExtAirRunning AT %IX."NirAdphos1".ExhAirRunning_2;
	::gNirAdphos.Status.Comms.Modules[1].iNirStatus AT %IW."NirAdphos1".NIRstatus_1;
	::gNirAdphos.Status.Comms.Modules[2].iNirStatus AT %IW."NirAdphos1".NIRstatus_2;
	::gNirAdphos.Status.Comms.Modules[1].TotalInFail AT %IB."NirAdphos1".EmFailNo_1;
	::gNirAdphos.Status.Comms.Modules[2].TotalInFail AT %IB."NirAdphos1".EmFailNo_2;
	::gNirAdphos.Signals.Out.xWatchDog AT %QX."NirAdphos1".WatchdogOut;
	::gNirAdphos.Status.Comms.Modules[1].AirPressIn AT %ID."NirAdphos1".airPressIn_1;
	::gNirAdphos.Status.Comms.Modules[1].AirPressOut AT %ID."NirAdphos1".airPressOut_1;
	::gNirAdphos.Status.Comms.Modules[1].SpeedIn AT %IW."NirAdphos1".actSpeedIn_1;
	::gNirAdphos.Status.Comms.Modules[1].SpeedOut AT %IW."NirAdphos1".actSpeedOut_1;
	::gNirAdphos.Status.Comms.Modules[1].Power AT %IW."NirAdphos1".actPower_1;
	::gNirAdphos.Status.Comms.Modules[1].AirFilter AT %IW."NirAdphos1".airFilter_1;
	::gNirAdphos.Status.Comms.Modules[2].AirPressIn AT %ID."NirAdphos1".airPressIn_2;
	::gNirAdphos.Status.Comms.Modules[2].AirPressOut AT %ID."NirAdphos1".airPressOut_2;
	::gNirAdphos.Status.Comms.Modules[2].AirFilter AT %IW."NirAdphos1".airFilter_2;
	::gNirAdphos.Status.Comms.Modules[2].SpeedIn AT %IW."NirAdphos1".actSpeedIn_2;
	::gNirAdphos.Status.Comms.Modules[2].SpeedOut AT %IW."NirAdphos1".actSpeedOut_2;
	::gNirAdphos.Status.Comms.Modules[2].Power AT %IW."NirAdphos1".actPower_2;
	::X20AI8321_207.Status01 AT %IB."X20AI8321_207".StatusInput01;
	::X20AI8321_207.Status02 AT %IB."X20AI8321_207".StatusInput02;
	::X20AT4222_209.Status01 AT %IB."X20AT4222_209".StatusInput01;
	::gInverterSignalsPowerLink[1].In.Hw.SerialNumber AT %ID."8I66xxxxxxx.0P-81".SerialNumber;
	::gInverterSignalsPowerLink[1].In.Hw.ModuleID AT %ID."8I66xxxxxxx.0P-81".ModuleID;
	::gInverterSignalsPowerLink[1].In.Hw.HwVariant AT %ID."8I66xxxxxxx.0P-81".HardwareVariant;
	::gInverterSignalsPowerLink[1].In.Hw.FwVersion AT %ID."8I66xxxxxxx.0P-81".FirmwareVersion;
	::gInverterSignalsPowerLink[1].In.Hw.ACPiSerialNumber AT %ID."8I66xxxxxxx.0P-81".ACPi_SerialNumber;
	::gInverterSignalsPowerLink[1].In.Hw.ACPiModuleID AT %ID."8I66xxxxxxx.0P-81".ACPi_ModuleID;
	::gInverterSignalsPowerLink[1].In.ActualSpeed AT %IW."8I66xxxxxxx.0P-81".RFRD_Input;
	::gInverterSignalsPowerLink[1].In.ActualTorque AT %IW."8I66xxxxxxx.0P-81".OTRN_Input;
	::gInverterSignalsPowerLink[1].In.ActualCurrent AT %IW."8I66xxxxxxx.0P-81".LCR_Input;
	::gInverterSignalsPowerLink[2].In.Hw.SerialNumber AT %ID."8I66xxxxxxx.0P-82".SerialNumber;
	::gInverterSignalsPowerLink[2].In.Hw.ModuleID AT %ID."8I66xxxxxxx.0P-82".ModuleID;
	::gInverterSignalsPowerLink[2].In.Hw.HwVariant AT %ID."8I66xxxxxxx.0P-82".HardwareVariant;
	::gInverterSignalsPowerLink[2].In.Hw.FwVersion AT %ID."8I66xxxxxxx.0P-82".FirmwareVersion;
	::gInverterSignalsPowerLink[2].In.ActualSpeed AT %IW."8I66xxxxxxx.0P-82".RFRD_Input;
	::gInverterSignalsPowerLink[2].In.ActualTorque AT %IW."8I66xxxxxxx.0P-82".OTRN_Input;
	::gInverterSignalsPowerLink[2].In.ActualCurrent AT %IW."8I66xxxxxxx.0P-82".LCR_Input;
	::gInverterSignalsPowerLink[2].In.Hw.ACPiSerialNumber AT %ID."8I66xxxxxxx.0P-82".ACPi_SerialNumber;
	::gInverterSignalsPowerLink[2].In.Hw.ACPiModuleID AT %ID."8I66xxxxxxx.0P-82".ACPi_ModuleID;
	::gDryerAnc.Inputs.xTransportMoving AT %IX."Printer".xRuningBelt;
	::gDryerAnc.Outputs.xRunTransport AT %QX."Printer".xRunTransport;
	::gDryerAnc.Outputs.xPrepareToDry AT %QX."Printer".xPrepareToDry;
	::gDryerAnc.Outputs.xStartDrying AT %QX."Printer".xStartDrying;
	::gDryerAnc.Inputs.xDrying AT %IX."Printer".xDrying;
	::gDryerAnc.Inputs.xReadyToDry AT %IX."Printer".xReadyToDry;
	::gDryerAnc.Inputs.xJamDetection AT %IX."Printer".xJamDetection;
	::gDryerAnc.Inputs.xTransportMoving AT %IX."Printer".xTransportMoving;
	::gDryerAnc.Inputs.xInRemote AT %IX."Printer".xInRemote;
	::gDryerAnc.Inputs.xReadyToEmptyBelt AT %IX."Printer".xReadyToEmptyBelt;
	::gDryerAnc.Parameters.rSpeedSetPoint AT %QD."Printer".rBeltSpeedSetPoint;
	::gDryerAnc.Parameters.rMediaLength AT %QD."Printer".rBoardLength;
	::gDryerAnc.Parameters.rMediaWidth AT %QD."Printer".rBoardWidth;
	::gDryerAnc.Parameters.rMediaThickness AT %QD."Printer".rBoardThickness;
	::gDryerAnc.Parameters.rMediaGap AT %QD."Printer".rBoardGap;
	::gDryerRemoteData.Signals.xMediaPresent AT %QX."Printer".Signals_xMediaPresent;
	::gDryerRemoteData.Signals.xBreakerOKBlowerInput AT %QX."Printer".Signals_xBreakerOKBlowerInput;
	::gDryerRemoteData.Signals.xBreakerOKBlowerOutput AT %QX."Printer".Signals_xBreakerOKBlowerOutput;
	::gDryerRemoteData.Signals.Safety.xMovementsEnabled AT %QX."Printer".Signals_Safety_xMovementsEnabled;
	::gDryerRemoteData.Signals.Safety.xRemoteEStopOK AT %QX."Printer".Signals_Safety_xRemoteEStopOK;
	::gDryerRemoteData.Signals.Safety.xEStopFrontOK AT %QX."Printer".Signals_Safety_xEStopFrontOK;
	::gDryerRemoteData.Signals.Safety.xEStopRearOK AT %QX."Printer".Signals_Safety_xEStopRearOK;
	::gDryerRemoteData.Signals.Safety.xClosedFrontInput AT %QX."Printer".Signals_Safety_xClosedFrontIn;
	::gDryerRemoteData.Signals.Safety.xClosedFrontOutput AT %QX."Printer".Signals_Safety_xClosedFrontOut;
	::gDryerRemoteData.Signals.Safety.xClosedRearInput AT %QX."Printer".Signals_Safety_xClosedRearIn;
	::gDryerRemoteData.Signals.Safety.xClosedRearOutput AT %QX."Printer".Signals_Safety_xClosedRearOut;
	::gDryerRemoteData.Signals.xMediaPresent AT %IX."Printer".Signals_xMediaPresent;
	::gDryerRemoteData.Signals.xBreakerOKBlowerInput AT %IX."Printer".Signals_xBreakerOKBlowerInput;
	::gDryerRemoteData.Signals.xBreakerOKBlowerOutput AT %IX."Printer".Signals_xBreakerOKBlowerOutput;
	::gDryerRemoteData.Signals.Safety.xMovementsEnabled AT %IX."Printer".Signals_Safety_xMovementsEnabled;
	::gDryerRemoteData.Signals.Safety.xRemoteEStopOK AT %IX."Printer".Signals_Safety_xRemoteEStopOK;
	::gDryerRemoteData.Signals.Safety.xEStopFrontOK AT %IX."Printer".Signals_Safety_xEStopFrontOK;
	::gDryerRemoteData.Signals.Safety.xEStopRearOK AT %IX."Printer".Signals_Safety_xEStopRearOK;
	::gDryerRemoteData.Signals.Safety.xClosedFrontInput AT %IX."Printer".Signals_Safety_xClosedFrontIn;
	::gDryerRemoteData.Signals.Safety.xClosedFrontOutput AT %IX."Printer".Signals_Safety_xClosedFrontOut;
	::gDryerRemoteData.Signals.Safety.xClosedRearInput AT %IX."Printer".Signals_Safety_xClosedRearIn;
	::gDryerRemoteData.Signals.Safety.xClosedRearOutput AT %IX."Printer".Signals_Safety_xClosedRearOut;
	::gDryerRemoteData.Commands.xRunTransport AT %IX."Printer".xRunTransport;
	::gDryerRemoteData.Commands.xPrepareToDry AT %IX."Printer".xPrepareToDry;
	::gDryerRemoteData.Commands.xStartDrying AT %IX."Printer".xStartDrying;
	::gDryerRemoteData.Parameters.rBeltSpeedSetPoint AT %ID."Printer".rBeltSpeedSetPoint;
	::gDryerRemoteData.Parameters.Media.rLength AT %ID."Printer".rBoardLength;
	::gDryerRemoteData.Parameters.Media.rWidth AT %ID."Printer".rBoardWidth;
	::gDryerRemoteData.Parameters.Media.rThickness AT %ID."Printer".rBoardThickness;
	::gDryerRemoteData.Parameters.xEnableNir AT %IX."Printer".xEnableNir;
	::gDryerRemoteData.Parameters.xEnableArcLamp AT %IX."Printer".xEnableArcLampDrying;
	::gDryerRemoteData.xCommsOK AT %IX."Printer".ModuleOk;
	::gNirAdphos.Status.xCommsOK AT %IX."NirAdphos1".ModuleOk;
	::gDryerRemoteData.Parameters.Media.rDocWidth AT %ID."Printer".rDocumentWidth;
	::gDryerRemoteData.Parameters.Media.rDocLength AT %ID."Printer".rDocumentLength;
	::gInverterSignalsPowerLink[1].In.AnalogInput[0] AT %IW."8I66xxxxxxx.0P-81".AI1R_Input;
	::gInverterSignalsPowerLink[1].In.AnalogInput[1] AT %IW."8I66xxxxxxx.0P-81".AI2R_Input;
	::gInverterSignalsPowerLink[1].In.AnalogInput[2] AT %IW."8I66xxxxxxx.0P-81".AI3R_Input;
	::gInverterSignalsPowerLink[1].In.DigitalInput[0] AT %IX."8I66xxxxxxx.0P-81".IL1R_Input_DI1;
	::gInverterSignalsPowerLink[1].In.DigitalInput[1] AT %IX."8I66xxxxxxx.0P-81".IL1R_Input_DI2;
	::gInverterSignalsPowerLink[1].In.DigitalInput[2] AT %IX."8I66xxxxxxx.0P-81".IL1R_Input_DI3;
	::gInverterSignalsPowerLink[1].In.DigitalInput[3] AT %IX."8I66xxxxxxx.0P-81".IL1R_Input_DI4;
	::gInverterSignalsPowerLink[1].In.DigitalInput[4] AT %IX."8I66xxxxxxx.0P-81".IL1R_Input_DI5;
	::gInverterSignalsPowerLink[1].In.DigitalInput[5] AT %IX."8I66xxxxxxx.0P-81".IL1R_Input_DI6;
	::gInverterSignalsPowerLink[1].In.DigitalInput[6] AT %IX."8I66xxxxxxx.0P-81".IL1R_Input_DAI1;
	::gInverterSignalsPowerLink[1].In.DigitalInput[7] AT %IX."8I66xxxxxxx.0P-81".IL1R_Input_DAI2;
	::gInverterSignalsPowerLink[1].Out.AnalogOutput AT %QW."8I66xxxxxxx.0P-81".AO1R_Output;
	::gInverterSignalsPowerLink[1].Out.DigitalOutput[0] AT %QX."8I66xxxxxxx.0P-81".OL1R_Output_R1;
	::gInverterSignalsPowerLink[1].Out.DigitalOutput[1] AT %QX."8I66xxxxxxx.0P-81".OL1R_Output_R2;
	::gInverterSignalsPowerLink[1].Out.DigitalOutput[2] AT %QX."8I66xxxxxxx.0P-81".OL1R_Output_DQ1;
	::gInverterSignalsPowerLink[2].In.AnalogInput[0] AT %IW."8I66xxxxxxx.0P-82".AI1R_Input;
	::gInverterSignalsPowerLink[2].In.AnalogInput[1] AT %IW."8I66xxxxxxx.0P-82".AI2R_Input;
	::gInverterSignalsPowerLink[2].In.AnalogInput[2] AT %IW."8I66xxxxxxx.0P-82".AI3R_Input;
	::gInverterSignalsPowerLink[2].In.DigitalInput[0] AT %IX."8I66xxxxxxx.0P-82".IL1R_Input_DI1;
	::gInverterSignalsPowerLink[2].In.DigitalInput[1] AT %IX."8I66xxxxxxx.0P-82".IL1R_Input_DI2;
	::gInverterSignalsPowerLink[2].In.DigitalInput[2] AT %IX."8I66xxxxxxx.0P-82".IL1R_Input_DI3;
	::gInverterSignalsPowerLink[2].In.DigitalInput[3] AT %IX."8I66xxxxxxx.0P-82".IL1R_Input_DI4;
	::gInverterSignalsPowerLink[2].In.DigitalInput[4] AT %IX."8I66xxxxxxx.0P-82".IL1R_Input_DI5;
	::gInverterSignalsPowerLink[2].In.DigitalInput[5] AT %IX."8I66xxxxxxx.0P-82".IL1R_Input_DI6;
	::gInverterSignalsPowerLink[2].In.DigitalInput[6] AT %IX."8I66xxxxxxx.0P-82".IL1R_Input_DAI1;
	::gInverterSignalsPowerLink[2].In.DigitalInput[7] AT %IX."8I66xxxxxxx.0P-82".IL1R_Input_DAI2;
	::gInverterSignalsPowerLink[2].Out.AnalogOutput AT %QW."8I66xxxxxxx.0P-82".AO1R_Output;
	::gInverterSignalsPowerLink[2].Out.DigitalOutput[0] AT %QX."8I66xxxxxxx.0P-82".OL1R_Output_R1;
	::gInverterSignalsPowerLink[2].Out.DigitalOutput[1] AT %QX."8I66xxxxxxx.0P-82".OL1R_Output_R2;
	::gInverterSignalsPowerLink[2].Out.DigitalOutput[2] AT %QX."8I66xxxxxxx.0P-82".OL1R_Output_DQ1;
	::gDryerRemoteData.Commands.xPrepareToEmptyBelt AT %IX."Printer".xPrepareToEmptyBelt;
	::gDryerRemoteData.Parameters.xLineEmptyingBelt AT %IX."Printer".xLineEmptyingBelt;
	::gDryerRemoteData.Parameters.Document.rOffsetL1 AT %IX."Printer".rDocumentOffsetL1;
	::gDryerRemoteData.Parameters.Document.rOffsetL2 AT %IX."Printer".rDocumentOffsetL2;
	::gDryerRemoteData.Parameters.Media.rDocCrossOffset AT %ID."Printer".rDocumentOffsetL1;
	::gDryerRemoteData.Parameters.rSubstratePowerReduction AT %ID."Printer".rSubstratePowerReduction;
	::gDryerRemoteData.Parameters.Document.rOffsetL1 AT %IX."Printer".rDocumentOffsetL1;
	::gInverterSignalsCanOpen[1].In.ActualCurrent AT %IW."ACPi_P66.01".LCR_3204_2002sub5;
	::gInverterSignalsCanOpen[1].In.ModuleOk AT %IX."ACPi_P66.01".ModuleOk;
	::gInverterSignalsCanOpen[1].Out.DigitalOutputs AT %QW."ACPi_P66.01".OL1R_5212_2016subd_Out;
	::gInverterSignalsCanOpen[1].In.DigitalInputs AT %IW."ACPi_P66.01".IL1R_5202_2016sub3;
	::gInverterSignalsCanOpen[1].In.AnalogInput[0] AT %IW."ACPi_P66.01".AI1R_5232_2016sub21;
	::gInverterSignalsCanOpen[1].In.AnalogInput[1] AT %IW."ACPi_P66.01".AI2R_5233_2016sub22;
	::gInverterSignalsCanOpen[1].Out.AnalogOutputSigned AT %QW."ACPi_P66.01".AO1R_5261_2016sub3e_Out;
	::gInverterSignalsCanOpen[1].In.ErrorID AT %IW."ACPi_P66.01".LFT_7121_2029sub16;
	::gInverterSignalsCanOpen[1].Out.ControlWord AT %QW."ACPi_P66.01".CMDD_8601_2038sub2_Out;
	::gInverterSignalsCanOpen[1].Out.SetSpeed AT %QW."ACPi_P66.01".LFRD_8602_2038sub3_Out;
	::gInverterSignalsCanOpen[1].In.StatusWord AT %IW."ACPi_P66.01".ETAD_8603_2038sub4;
	::gInverterSignalsCanOpen[1].In.ActualSpeed AT %IW."ACPi_P66.01".RFRD_8604_2038sub5;
	::gInverterSignalsCanOpen[1].Out.Acceleration AT %QW."ACPi_P66.01".ACC_9001_203csub2_Out;
	::gInverterSignalsCanOpen[1].Out.Deceleration AT %QW."ACPi_P66.01".DEC_9002_203csub3_Out;
	::gInverterSignalsCanOpen[1].In.ActualTorque AT %IW."ACPi_P66.01".TorqueActualValue_6077;
	::gInverterSignalsCanOpen[2].In.ModuleOk AT %IX."ACPi_P66.02".ModuleOk;
	::gInverterSignalsCanOpen[2].In.ActualCurrent AT %IW."ACPi_P66.02".LCR_3204_2002sub5;
	::gInverterSignalsCanOpen[2].In.DigitalInputs AT %IW."ACPi_P66.02".IL1R_5202_2016sub3;
	::gInverterSignalsCanOpen[2].Out.DigitalOutputs AT %QW."ACPi_P66.02".OL1R_5212_2016subd_Out;
	::gInverterSignalsCanOpen[2].In.AnalogInput[0] AT %IW."ACPi_P66.02".AI1R_5232_2016sub21;
	::gInverterSignalsCanOpen[2].In.AnalogInput[1] AT %IW."ACPi_P66.02".AI2R_5233_2016sub22;
	::gInverterSignalsCanOpen[2].Out.AnalogOutputSigned AT %QW."ACPi_P66.02".AO1R_5261_2016sub3e_Out;
	::gInverterSignalsCanOpen[2].In.ErrorID AT %IW."ACPi_P66.02".LFT_7121_2029sub16;
	::gInverterSignalsCanOpen[2].Out.ControlWord AT %QW."ACPi_P66.02".CMDD_8601_2038sub2_Out;
	::gInverterSignalsCanOpen[2].Out.SetSpeed AT %QW."ACPi_P66.02".LFRD_8602_2038sub3_Out;
	::gInverterSignalsCanOpen[2].In.StatusWord AT %IW."ACPi_P66.02".ETAD_8603_2038sub4;
	::gInverterSignalsCanOpen[2].In.ActualSpeed AT %IW."ACPi_P66.02".RFRD_8604_2038sub5;
	::gInverterSignalsCanOpen[2].Out.Acceleration AT %QW."ACPi_P66.02".ACC_9001_203csub2_Out;
	::gInverterSignalsCanOpen[2].Out.Deceleration AT %QW."ACPi_P66.02".DEC_9002_203csub3_Out;
	::gInverterSignalsCanOpen[2].In.ActualTorque AT %IW."ACPi_P66.02".TorqueActualValue_6077;
	::gNirAdphos.Status.xEnabledDDC AT %QX."NirAdphos1".Enable_DDC;
	::gDryerRemoteData.Parameters.Media.rDocCrossOffset AT %ID."Printer".rDocumentOffset;
	::gDryerRemoteData.Parameters.Media.rCrossOffset AT %ID."Printer".rCrossOffset;
	::gDryerRemoteData.Parameters.xEnableDDC AT %IX."Printer".xEnableDDC;
	::gDryerRemoteData.Parameters.xPrinterBeltRuning AT %IX."Printer".xPrinterBeltRuning;
END_VAR
```

### Acp10map.ncm - X20CP0483/Motion/Acp10map.ncm
```
NcMapping (NcSwId=Acp10, DisabledNodesAreHidden=False)
  NcObject gAxis01 (ModuleId=8EI044HWS10.xxxx-1_BELT, Type=ncAXIS, Channel=1, AcoposSimulation=Off, InitParameter=BeltS1400i, AcoposParameter=BeltS1400a, Disabled=FALSE, ModuleDisabled=FALSE)
  NcObject 8EI044HWS10.xxxx-1_ncV_AXIS1 (ModuleId=8EI044HWS10.xxxx-1_BELT, Type=ncV_AXIS, Channel=1, Disabled=TRUE, ModuleDisabled=FALSE)
  NcObject gAxis02 (ModuleId=8EI2X2MWS10.xxxx-1, Type=ncAXIS, Channel=1, AcoposSimulation=Off, InitParameter=BK1_S1400i, AcoposParameter=BK1_S1400a, Disabled=FALSE, ModuleDisabled=FALSE)
  NcObject 8EI4X5MWS10.xxxx-1_ncV_AXIS1 (ModuleId=8EI2X2MWS10.xxxx-1, Type=ncV_AXIS, Channel=1, Disabled=TRUE, ModuleDisabled=FALSE)
```

## Logical view

Binary libraries used (declarations not repeated): Acp10_MC 5.31.1, Acp10man 5.31.1, Acp10par 5.31.1, Acp10sdc 5.31.1, Acp10sim 5.31.1, ArProject, AsBrStr, AsCANopen, AsEPL, AsIecCon, AsIOAcc, AsMath, AsOpcUas, AsSafety, AsTCP, brsystem, ErrACS380, FileIO, IecCheck, MpAlarmX 5.24.6, MpCom 5.24.6, NcGlobal 5.31.1, operator, sys_lib, UtWs 2.01.0

- BatchCompile.bat (not shown)

- Project.language (not shown)

### Program Logical/AsSafetySolution/SafetySample (IEC) - Handling

- Visualisation Logical/AsSafetySolution/Panel (not shown)

- Data object Logical/AxisTables/AcpErrTxt (Ett) (no source held here)

### Data object Logical/AxisTables/Belt17000_i (Ax)

#### Belt1.ax
```
InitParameter (Version=5.21.2, NcSwId=ACP10)
  ACP10AXIS_typ:
    dig_in:
      level:
        reference = ncACTIV_LO
        pos_hw_end = ncACTIV_HI
        neg_hw_end = ncACTIV_HI
        trigger1 = ncACTIV_LO
        trigger2 = ncACTIV_LO
    encoder_if:
      parameter:
        count_dir = ncSTANDARD
        scaling:
          load:
            units = 1000
            rev_motor = 1
    limit:
      parameter:
        v_pos = 435800.0
        v_neg = 435800.0
        a1_pos = 1400000.0
        a2_pos = 1400000.0
        a1_neg = 1400000.0
        a2_neg = 1400000.0
        t_jolt = 0.0
        t_in_pos = 0.0
        pos_sw_end = 8388607
        neg_sw_end = -8388608
        ds_warning = 500.0
        ds_stop = 1000.0
        a_stop = 6.53E+07
        dv_stop = 0.0
        dv_stop_mode = ncOFF
    controller:
      mode = ncPOSITION
      position:
        kv = 414.0
        tn = 0.0
        t_predict = 0.0004
        t_total = 0.0004
        p_max = 1.0E+30
        i_max = 0.0
      speed:
        kv = 54.75
        tn = 0.0
        t_filter = 0.0
        isq_filter1:
          type = ncOFF
          a0 = 0.0
          a1 = 0.0
          b0 = 0.0
          b1 = 0.0
          b2 = 0.0
          c0_par_id = 0
          c1_par_id = 0
        isq_filter2:
          type = ncOFF
          a0 = 0.0
          a1 = 0.0
          b0 = 0.0
          b1 = 0.0
          b2 = 0.0
          c0_par_id = 0
          c1_par_id = 0
        isq_filter3:
          type = ncOFF
          a0 = 0.0
          a1 = 0.0
          b0 = 0.0
          b1 = 0.0
          b2 = 0.0
          c0_par_id = 0
          c1_par_id = 0
      uf:
        type = ncLINEAR
        auto_config = ncMOTOR_PAR
        u0 = 0.0
        un = 0.0
        fn = 50.0
        k_f_slip = 0.0
      ff:
        mode = ncSTANDARD
        torque_load = 0.0
        torque_pos = 0.0
        torque_neg = 0.0
        kv_torque = 0.0
        inertia = 0.0
        t_filter_a = 0.0
      fb:
        mode = ncSTANDARD
        speed_mix_ratio = 0.0
        speed_kv = 2.0
      model:
        mass1:
          inertia = 0.0
          viscous_friction = 0.0
        mass2:
          inertia = 0.0
          viscous_friction = 0.0
          stiffness = 0.0
          damping = 0.0
    move:
      stop:
        parameter[0]:
          decel_ramp = ncA_LIMIT
          controller = ncON
        parameter[1]:
          decel_ramp = ncA_LIMIT
          controller = ncON
        parameter[2]:
          decel_ramp = ncA_LIMIT
          controller = ncON
        parameter[3]:
          decel_ramp = ncA_LIMIT
          controller = ncON
        quickstop:
          decel_ramp = ncA_LIMIT
          t_jolt = 0.0
        drive_error:
          decel_ramp = ncA_LIMIT
      homing:
        parameter:
          s = 0
          v_switch = 5000.0
          v_trigger = 500.0
          a = 50000.0
          mode = ncDIRECT
          edge_sw = ncPOSITIVE
          start_dir = ncPOSITIVE
          trigg_dir = ncPOSITIVE
          ref_pulse = ncOFF
          fix_dir = ncOFF
          tr_s_block = 0.0
          torque_lim = 0.0
          ds_block = 0.0
          ds_stop = 0.0
      basis:
        parameter:
          v_pos = 5000.0
          v_neg = 5000.0
          a1_pos = 50000.0
          a2_pos = 50000.0
          a1_neg = 50000.0
          a2_neg = 50000.0
    message:
      text:
        parameter:
          format = ncBREAK
          columns = 80
          data_modul = acp10etxen
```

- Data object Logical/AxisTables/BeltP4_a (Apt) (no source held here)

### BeltI.ax
```
InitParameter (Version=5.12.2, NcSwId=ACP10)
  ACP10AXIS_typ:
    dig_in:
      level:
        reference = ncACTIV_LO
        pos_hw_end = ncACTIV_HI
        neg_hw_end = ncACTIV_HI
        trigger1 = ncACTIV_LO
        trigger2 = ncACTIV_LO
    encoder_if:
      parameter:
        count_dir = ncSTANDARD
        scaling:
          load:
            units = 1000
            rev_motor = 1
    limit:
      parameter:
        v_pos = 435800.0
        v_neg = 435800.0
        a1_pos = 653000.0
        a2_pos = 653000.0
        a1_neg = 653000.0
        a2_neg = 653000.0
        t_jolt = 0.0
        t_in_pos = 0.0
        pos_sw_end = 2000000000
        neg_sw_end = -2000000000
        ds_warning = 500.0
        ds_stop = 1000.0
        a_stop = 6.53E+07
        dv_stop = 0.0
        dv_stop_mode = ncOFF
    controller:
      mode = ncPOSITION
      position:
        kv = 840.0
        tn = 0.0
        t_predict = 0.0004
        t_total = 0.0004
        p_max = 1.0E+30
        i_max = 0.0
      speed:
        kv = 4.4
        tn = 0.0
        t_filter = 0.0
        isq_filter1:
          type = ncOFF
          a0 = 0.0
          a1 = 0.0
          b0 = 0.0
          b1 = 0.0
          b2 = 0.0
          c0_par_id = 0
          c1_par_id = 0
        isq_filter2:
          type = ncOFF
          a0 = 0.0
          a1 = 0.0
          b0 = 0.0
          b1 = 0.0
          b2 = 0.0
          c0_par_id = 0
          c1_par_id = 0
        isq_filter3:
          type = ncOFF
          a0 = 0.0
          a1 = 0.0
          b0 = 0.0
          b1 = 0.0
          b2 = 0.0
          c0_par_id = 0
          c1_par_id = 0
      uf:
        type = ncLINEAR
        auto_config = ncMOTOR_PAR
        u0 = 0.0
        un = 0.0
        fn = 50.0
        k_f_slip = 0.0
      ff:
        mode = ncSTANDARD
        torque_load = 0.0
        torque_pos = 0.0
        torque_neg = 0.0
        kv_torque = 0.0
        inertia = 0.0
        t_filter_a = 0.0
      fb:
        mode = ncSTANDARD
        speed_mix_ratio = 0.0
        speed_kv = 2.0
      model:
        mass1:
          inertia = 0
          viscous_friction = 0
        mass2:
          inertia = 0
          viscous_friction = 0
          stiffness = 0
          damping = 0
    move:
      stop:
        parameter[0]:
          decel_ramp = ncA_LIMIT
          controller = ncON
        parameter[1]:
          decel_ramp = ncA_LIMIT
          controller = ncON
        parameter[2]:
          decel_ramp = ncA_LIMIT
          controller = ncON
        parameter[3]:
          decel_ramp = ncA_LIMIT
          controller = ncON
        quickstop:
          decel_ramp = ncA_LIMIT
          t_jolt = 0.0
        drive_error:
          decel_ramp = ncA_LIMIT
      homing:
        parameter:
          s = 0
          v_switch = 5000.0
          v_trigger = 500.0
          a = 50000.0
          mode = ncDIRECT
          edge_sw = ncPOSITIVE
          start_dir = ncPOSITIVE
          trigg_dir = ncPOSITIVE
          ref_pulse = ncOFF
          fix_dir = ncOFF
          tr_s_block = 0.0
          torque_lim = 0.0
          ds_block = 0.0
          ds_stop = 0.0
      basis:
        parameter:
          v_pos = 5000.0
          v_neg = 5000.0
          a1_pos = 50000.0
          a2_pos = 50000.0
          a1_neg = 50000.0
          a2_neg = 50000.0
    message:
      text:
        parameter:
          format = ncBREAK
          columns = 80
          data_modul = acp10etxen
```

- Data object Logical/AxisTables/BeltP5_a (Apt) (no source held here)

### BeltA.apt
```
AcoposParameterTable:
  Root Parameters:
    128 = 1 (Name=SGEN_SW_END_IGNORE)  // Limit values: Ignore SW end positions
```

### BeltI.ax
```
InitParameter (Version=5.15.1, NcSwId=ACP10)
  ACP10AXIS_typ:
    dig_in:
      level:
        reference = ncACTIV_LO
        pos_hw_end = ncACTIV_HI
        neg_hw_end = ncACTIV_HI
        trigger1 = ncACTIV_LO
        trigger2 = ncACTIV_LO
    encoder_if:
      parameter:
        count_dir = ncSTANDARD
        scaling:
          load:
            units = 1000
            rev_motor = 1
    limit:
      parameter:
        v_pos = 435800.0
        v_neg = 435800.0
        a1_pos = 1400000.0  // Acceleration in positive direction. Previous 653000.0
        a2_pos = 1400000.0
        a1_neg = 1400000.0
        a2_neg = 1400000.0
        t_jolt = 0.0
        t_in_pos = 0.0
        pos_sw_end = 2000000000
        neg_sw_end = -2000000000
        ds_warning = 500.0
        ds_stop = 1000.0
        a_stop = 6.53E+07
        dv_stop = 0.0
        dv_stop_mode = ncOFF
    controller:
      mode = ncPOSITION
      position:
        kv = 414.0
        tn = 0.0
        t_predict = 0.0004
        t_total = 0.0004
        p_max = 1.0E+30
        i_max = 0.0
      speed:
        kv = 54.75
        tn = 0.0
        t_filter = 0.0
        isq_filter1:
          type = ncOFF
          a0 = 0.0
          a1 = 0.0
          b0 = 0.0
          b1 = 0.0
          b2 = 0.0
          c0_par_id = 0
          c1_par_id = 0
        isq_filter2:
          type = ncOFF
          a0 = 0.0
          a1 = 0.0
          b0 = 0.0
          b1 = 0.0
          b2 = 0.0
          c0_par_id = 0
          c1_par_id = 0
        isq_filter3:
          type = ncOFF
          a0 = 0.0
          a1 = 0.0
          b0 = 0.0
          b1 = 0.0
          b2 = 0.0
          c0_par_id = 0
          c1_par_id = 0
      uf:
        type = ncLINEAR
        auto_config = ncMOTOR_PAR
        u0 = 0.0
        un = 0.0
        fn = 50.0
        k_f_slip = 0.0
      ff:
        mode = ncSTANDARD
        torque_load = 0.0
        torque_pos = 0.0
        torque_neg = 0.0
        kv_torque = 0.0
        inertia = 0.0
        t_filter_a = 0.0
      fb:
        mode = ncSTANDARD
        speed_mix_ratio = 0.0
        speed_kv = 2.0
      model:
        mass1:
          inertia = 0
          viscous_friction = 0
        mass2:
          inertia = 0
          viscous_friction = 0
          stiffness = 0
          damping = 0
    move:
      stop:
        parameter[0]:
          decel_ramp = ncA_LIMIT
          controller = ncON
        parameter[1]:
          decel_ramp = ncA_LIMIT
          controller = ncON
        parameter[2]:
          decel_ramp = ncA_LIMIT
          controller = ncON
        parameter[3]:
          decel_ramp = ncA_LIMIT
          controller = ncON
        quickstop:
          decel_ramp = ncA_LIMIT
          t_jolt = 0.0
        drive_error:
          decel_ramp = ncA_LIMIT
      homing:
        parameter:
          s = 0
          v_switch = 5000.0
          v_trigger = 500.0
          a = 50000.0
          mode = ncDIRECT
          edge_sw = ncPOSITIVE
          start_dir = ncPOSITIVE
          trigg_dir = ncPOSITIVE
          ref_pulse = ncOFF
          fix_dir = ncOFF
          tr_s_block = 0.0
          torque_lim = 0.0
          ds_block = 0.0
          ds_stop = 0.0
      basis:
        parameter:
          v_pos = 5000.0
          v_neg = 5000.0
          a1_pos = 50000.0
          a2_pos = 50000.0
          a1_neg = 50000.0
          a2_neg = 50000.0
    message:
      text:
        parameter:
          format = ncBREAK
          columns = 80
          data_modul = acp10etxen
```

### BeltI.ax
```
InitParameter (Version=5.02.1, NcSwId=Acp10)
  ACP10AXIS_typ:
    dig_in:
      level:
        reference = ncACTIV_LO
        pos_hw_end = ncACTIV_HI
        neg_hw_end = ncACTIV_HI
        trigger1 = ncACTIV_LO
        trigger2 = ncACTIV_LO
    encoder_if:
      parameter:
        count_dir = ncSTANDARD
        scaling:
          load:
            units = 1000
            rev_motor = 1
    limit:
      parameter:
        v_pos = 435800.0
        v_neg = 435800.0
        a1_pos = 653000.0
        a2_pos = 653000.0
        a1_neg = 653000.0
        a2_neg = 653000.0
        t_jolt = 0
        t_in_pos = 0
        pos_sw_end = 8388607
        neg_sw_end = -8388608
        ds_warning = 500.0
        ds_stop = 1000.0
        a_stop = 6.53E+07
        dv_stop = 0
        dv_stop_mode = ncOFF
    controller:
      mode = ncPOSITION
      position:
        kv = 661.0
        tn = 0
        t_predict = 0.0004
        t_total = 0.0004
        p_max = 1.0e30
        i_max = 0
      speed:
        kv = 0.5
        tn = 0
        t_filter = 0.0
        isq_filter1:
          type = ncNOTCH
          a0 = 1878.67
          a1 = 400.0
          b0 = 0.0
          b1 = 0.0
          b2 = 0.0
          c0_par_id = 0
          c1_par_id = 0
        isq_filter2:
          type = ncOFF
          a0 = 2495.11
          a1 = 400.0
          b0 = 0.0
          b1 = 0.0
          b2 = 0.0
          c0_par_id = 0
          c1_par_id = 0
        isq_filter3:
          type = ncOFF
          a0 = 0.0
          a1 = 0.0
          b0 = 0.0
          b1 = 0.0
          b2 = 0.0
          c0_par_id = 0
          c1_par_id = 0
      uf:
        type = ncLINEAR
        auto_config = ncMOTOR_PAR
        u0 = 0
        un = 0
        fn = 50.0
        k_f_slip = 0
      ff:
        torque_load = 0.0
        torque_pos = 0.0
        torque_neg = 0.0
        kv_torque = 0.0
        inertia = 0.0
        t_filter_a = 0.0
    move:
      stop:
        parameter[0]:
          decel_ramp = ncA_LIMIT
          controller = ncON
        parameter[1]:
          decel_ramp = ncA_LIMIT
          controller = ncON
        parameter[2]:
          decel_ramp = ncA_LIMIT
          controller = ncON
        parameter[3]:
          decel_ramp = ncA_LIMIT
          controller = ncON
        quickstop:
          decel_ramp = ncA_LIMIT
          t_jolt = 0
        drive_error:
          decel_ramp = ncA_LIMIT
      homing:
        parameter:
          s = 0
          v_switch = 5000
          v_trigger = 500
          a = 50000
          mode = ncDIRECT
          edge_sw = ncPOSITIVE
          start_dir = ncPOSITIVE
          trigg_dir = ncPOSITIVE
          ref_pulse = ncOFF
          fix_dir = ncOFF
          tr_s_block = 0
          torque_lim = 0
          ds_block = 0
          ds_stop = 0
      basis:
        parameter:
          v_pos = 5000
          v_neg = 5000
          a1_pos = 50000
          a2_pos = 50000
          a1_neg = 50000
          a2_neg = 50000
    message:
      text:
        parameter:
          format = ncBREAK
          columns = 80
          data_modul = acp10etxen
```

- Data object Logical/AxisTables/BK1_Cube_a (Apt) (no source held here)

### Data object Logical/AxisTables/BK1_i (Ax)

#### BK1_i.ax
```
InitParameter (Version=5.11.1, NcSwId=ACP10)
  ACP10AXIS_typ:
    dig_in:
      level:
        reference = ncACTIV_LO
        pos_hw_end = ncACTIV_HI
        neg_hw_end = ncACTIV_HI
        trigger1 = ncACTIV_HI
        trigger2 = ncACTIV_HI
    encoder_if:
      parameter:
        count_dir = ncSTANDARD
        scaling:
          load:
            units = 1000
            rev_motor = 1
    limit:
      parameter:
        v_pos = 60050.0
        v_neg = 60050.0
        a1_pos = 725000.0
        a2_pos = 725000.0
        a1_neg = 725000.0
        a2_neg = 725000.0
        t_jolt = 0.0
        t_in_pos = 0.0
        pos_sw_end = 700000
        neg_sw_end = -700000
        ds_warning = 500.0
        ds_stop = 1000.0
        a_stop = 725000.0
        dv_stop = 0.0
        dv_stop_mode = ncOFF
    controller:
      mode = ncPOSITION
      position:
        kv = 160.0
        tn = 0.0
        t_predict = 0.0004
        t_total = 0.0004
        p_max = 1.0E+30
        i_max = 0.0
      speed:
        kv = 1.15
        tn = 0.0
        t_filter = 0.0
        isq_filter1:
          type = ncOFF
          a0 = 0.0
          a1 = 0.0
          b0 = 0.0
          b1 = 0.0
          b2 = 0.0
          c0_par_id = 0
          c1_par_id = 0
        isq_filter2:
          type = ncOFF
          a0 = 0.0
          a1 = 0.0
          b0 = 0.0
          b1 = 0.0
          b2 = 0.0
          c0_par_id = 0
          c1_par_id = 0
        isq_filter3:
          type = ncOFF
          a0 = 0.0
          a1 = 0.0
          b0 = 0.0
          b1 = 0.0
          b2 = 0.0
          c0_par_id = 0
          c1_par_id = 0
      uf:
        type = ncLINEAR
        auto_config = ncMOTOR_PAR
        u0 = 0.0
        un = 0.0
        fn = 50.0
        k_f_slip = 0.0
      ff:
        mode = ncSTANDARD
        torque_load = 0.0
        torque_pos = 0.0
        torque_neg = 0.0
        kv_torque = 0.0
        inertia = 0.0
        t_filter_a = 0.0
      fb:
        mode = ncSTANDARD
        speed_mix_ratio = 0.0
        speed_kv = 2.0
      model:
        mass1:
          inertia = 0
          viscous_friction = 0
        mass2:
          inertia = 0
          viscous_friction = 0
          stiffness = 0
          damping = 0
    move:
      stop:
        parameter[0]:
          decel_ramp = ncA_LIMIT
          controller = ncON
        parameter[1]:
          decel_ramp = ncA_LIMIT
          controller = ncON
        parameter[2]:
          decel_ramp = ncA_LIMIT
          controller = ncON
        parameter[3]:
          decel_ramp = ncA_LIMIT
          controller = ncON
        quickstop:
          decel_ramp = ncA_LIMIT
          t_jolt = 0.0
        drive_error:
          decel_ramp = ncA_LIMIT
      homing:
        parameter:
          s = 23200
          v_switch = 5000.0
          v_trigger = 500.0
          a = 50000.0
          mode = ncABS_SWITCH
          edge_sw = ncPOSITIVE
          start_dir = ncNEGATIVE
          trigg_dir = ncNEGATIVE
          ref_pulse = ncOFF
          fix_dir = ncOFF
          tr_s_block = 0.0
          torque_lim = 0.0
          ds_block = 0.0
          ds_stop = 0.0
      basis:
        parameter:
          v_pos = 5000.0
          v_neg = 5000.0
          a1_pos = 50000.0
          a2_pos = 50000.0
          a1_neg = 50000.0
          a2_neg = 50000.0
    message:
      text:
        parameter:
          format = ncBREAK
          columns = 80
          data_modul = acp10etxen
```

### BK1_a.apt
```
AcoposParameterTable:
  Root Parameters:
    944 = STAT_TRIGGER1 (Name=REFERENCE_SWITCH_PARID)  // Digital inputs: Parameter ID for reference switch
    10 = 47 (Name=R_BLEEDER_EXT, Unit=Ohm)  // Bleeder: External: Resistance
    11 = 300 (Name=TEMP_MAX_BLEEDER_EXT, Unit=°C)  // Bleeder: External: Limit temperature
    12 = 1.4 (Name=RTH_BLEEDER_AMB_EXT, Unit=K/W)  // Bleeder: External: Thermal resistance
    13 = 30.82 (Name=CTH_BLEEDER_EXT, Unit=Ws/K)  // Bleeder: External: Thermal capacity
    398 = 1 (Name=BLEEDER_SELECTOR_EXT)  // Bleeder: Selector
```

- Data object Logical/AxisTables/BK_17000_i (Ax) (no source held here)

### BK_sim_a.apt
```
AcoposParameterTable:
  Root Parameters:
    777 = 4096 (Name=FUNCTION_BLOCK_CREATE)  // Function block: Create a FB instance
    944 = 4096 (Name=REFERENCE_SWITCH_PARID)  // Digital inputs: Parameter ID for reference switch
    VAR:
      4096 = 1 (Name=VAR_I4_0+0)  // FB0 VAR I4 variable0
```

### Data object Logical/AxisTables/NonCrash_i (Ax)

#### NonCrash_i.ax
```
InitParameter (Version=5.02.1, NcSwId=ACP10)
  ACP10AXIS_typ:
    dig_in:
      level:
        reference = ncACTIV_LO
        pos_hw_end = ncACTIV_HI
        neg_hw_end = ncACTIV_HI
        trigger1 = ncACTIV_LO
        trigger2 = ncACTIV_LO
    encoder_if:
      parameter:
        count_dir = ncSTANDARD
        scaling:
          load:
            units = 1000
            rev_motor = 1
    limit:
      parameter:
        v_pos = 435800.0
        v_neg = 435800.0
        a1_pos = 653000.0
        a2_pos = 653000.0
        a1_neg = 653000.0
        a2_neg = 653000.0
        t_jolt = 0.0
        t_in_pos = 0.0
        pos_sw_end = 8388607
        neg_sw_end = -8388608
        ds_warning = 500.0
        ds_stop = 1000.0
        a_stop = 6.53E+07
        dv_stop = 0.0
        dv_stop_mode = ncOFF
    controller:
      mode = ncPOSITION
      position:
        kv = 508.0
        tn = 0.0
        t_predict = 0.0004
        t_total = 0.0004
        p_max = 1.0E+30
        i_max = 0.0
      speed:
        kv = 0.15
        tn = 0.0
        t_filter = 0.0
        isq_filter1:
          type = ncOFF
          a0 = 0.0
          a1 = 0.0
          b0 = 0.0
          b1 = 0.0
          b2 = 0.0
          c0_par_id = 0
          c1_par_id = 0
        isq_filter2:
          type = ncOFF
          a0 = 0.0
          a1 = 0.0
          b0 = 0.0
          b1 = 0.0
          b2 = 0.0
          c0_par_id = 0
          c1_par_id = 0
        isq_filter3:
          type = ncOFF
          a0 = 0.0
          a1 = 0.0
          b0 = 0.0
          b1 = 0.0
          b2 = 0.0
          c0_par_id = 0
          c1_par_id = 0
      uf:
        type = ncLINEAR
        auto_config = ncMOTOR_PAR
        u0 = 0.0
        un = 0.0
        fn = 50.0
        k_f_slip = 0.0
      ff:
        torque_load = 0.0
        torque_pos = 0.0
        torque_neg = 0.0
        kv_torque = 0.0
        inertia = 0.0
        t_filter_a = 0.0
    move:
      stop:
        parameter[0]:
          decel_ramp = ncA_LIMIT
          controller = ncON
        parameter[1]:
          decel_ramp = ncA_LIMIT
          controller = ncON
        parameter[2]:
          decel_ramp = ncA_LIMIT
          controller = ncON
        parameter[3]:
          decel_ramp = ncA_LIMIT
          controller = ncON
        quickstop:
          decel_ramp = ncA_LIMIT
          t_jolt = 0.0
        drive_error:
          decel_ramp = ncA_LIMIT
      homing:
        parameter:
          s = 0
          v_switch = 5000.0
          v_trigger = 500.0
          a = 50000.0
          mode = ncDIRECT
          edge_sw = ncPOSITIVE
          start_dir = ncPOSITIVE
          trigg_dir = ncPOSITIVE
          ref_pulse = ncOFF
          fix_dir = ncOFF
          tr_s_block = 0.0
          torque_lim = 0.0
          ds_block = 0.0
          ds_stop = 0.0
      basis:
        parameter:
          v_pos = 5000.0
          v_neg = 5000.0
          a1_pos = 50000.0
          a2_pos = 50000.0
          a1_neg = 50000.0
          a2_neg = 50000.0
    message:
      text:
        parameter:
          format = ncBREAK
          columns = 80
          data_modul = acp10etxen
```

- Data object Logical/AxisTables/SM_a (Apt) (no source held here)
